SPLINE
SPL {X  -158.491, Y  +370.077, Z    +0.000, E1   +15.910, E3 +25237.550}
SPL {X  -159.771, Y  +383.450, Z    +0.000, E1    +6.314, E3 +25260.705}
SPL {X  -160.000, Y  +392.463, Z    +0.000, E1    +0.112, E3 +25267.212}
SPL {X  -160.000, Y  +399.874, Z    +0.000, E1    -5.508, E3 +25271.714}
SPL {X  -160.000, Y  +411.622, Z    +0.000, E1   -13.815, E3 +25283.834}
SPL {X  -160.000, Y  +419.836, Z    +0.000, E1   -18.198, E3 +25299.008}
SPL {X  -160.000, Y  +430.523, Z    +0.000, E1   -21.710, E3 +25329.208}
SPL {X  -160.000, Y  +433.426, Z    +0.000, E1   -21.735, E3 +25344.623}
SPL {X  -160.000, Y  +436.131, Z    +0.000, E1   -21.710, E3 +25359.098}
SPL {X  -160.000, Y  +439.046, Z    +0.000, E1   -21.732, E3 +25374.591}
SPL {X  -160.000, Y  +442.009, Z    +0.000, E1   -21.719, E3 +25390.413}
SPL {X  -160.000, Y  +444.891, Z    +0.000, E1   -21.724, E3 +25405.769}
SPL {X  -160.000, Y  +449.017, Z    +0.000, E1   -21.792, E3 +25427.560}
SPL {X  -160.000, Y  +452.864, Z    +0.000, E1   -21.730, E3 +25448.178}
SPL {X  -160.000, Y  +455.470, Z    +0.000, E1   -21.722, E3 +25462.067}
SPL {X  -160.000, Y  +458.295, Z    +0.000, E1   -21.738, E3 +25477.088}
SPL {X  -160.000, Y  +461.133, Z    +0.000, E1   -21.720, E3 +25492.271}
SPL {X  -160.000, Y  +464.458, Z    +0.000, E1   -21.770, E3 +25509.789}
SPL {X  -160.000, Y  +468.250, Z    +0.000, E1   -21.764, E3 +25529.943}
SPL {X  -160.000, Y  +472.226, Z    +0.000, E1   -21.782, E3 +25551.101}
SPL {X  -160.000, Y  +476.333, Z    +0.000, E1   -21.767, E3 +25573.015}
SPL {X  -160.000, Y  +480.244, Z    +0.000, E1   -21.765, E3 +25593.880}
SPL {X  -160.000, Y  +484.301, Z    +0.000, E1   -21.775, E3 +25615.408}
SPL {X  -160.000, Y  +488.201, Z    +0.000, E1   -21.768, E3 +25636.168}
SPL {X  -160.000, Y  +492.394, Z    +0.000, E1   -21.802, E3 +25658.343}
SPL {X  -160.000, Y  +496.781, Z    +0.000, E1   -21.798, E3 +25681.654}
SPL {X  -160.000, Y  +501.083, Z    +0.000, E1   -21.796, E3 +25704.584}
SPL {X  -160.000, Y  +504.917, Z    +0.000, E1   -21.764, E3 +25725.088}
SPL {X  -160.000, Y  +508.886, Z    +0.000, E1   -21.791, E3 +25746.174}
SPL {X  -160.000, Y  +513.057, Z    +0.000, E1   -21.767, E3 +25768.482}
SPL {X  -160.000, Y  +517.221, Z    +0.000, E1   -21.778, E3 +25790.635}
SPL {X  -160.000, Y  +521.677, Z    +0.000, E1   -21.781, E3 +25814.396}
SPL {X  -160.000, Y  +525.729, Z    +0.000, E1   -21.753, E3 +25836.035}
SPL {X  -160.000, Y  +529.456, Z    +0.000, E1   -21.766, E3 +25855.815}
SPL {X  -160.000, Y  +533.608, Z    +0.000, E1   -21.776, E3 +25877.945}
SPL {X  -160.000, Y  +538.227, Z    +0.000, E1   -21.794, E3 +25902.477}
SPL {X  -160.000, Y  +542.483, Z    +0.000, E1   -21.764, E3 +25925.203}
SPL {X  -160.000, Y  +546.194, Z    +0.000, E1   -21.754, E3 +25945.019}
SPL {X  -160.000, Y  +550.131, Z    +0.000, E1   -21.771, E3 +25965.955}
SPL {X  -160.000, Y  +554.462, Z    +0.000, E1   -21.777, E3 +25989.009}
SPL {X  -160.000, Y  +558.542, Z    +0.000, E1   -21.758, E3 +26010.782}
SPL {X  -160.000, Y  +562.615, Z    +0.000, E1   -21.776, E3 +26032.437}
SPL {X  -160.000, Y  +566.764, Z    +0.000, E1   -21.764, E3 +26054.562}
SPL {X  -160.000, Y  +570.657, Z    +0.000, E1   -21.758, E3 +26075.310}
SPL {X  -160.000, Y  +574.688, Z    +0.000, E1   -21.771, E3 +26096.752}
SPL {X  -160.000, Y  +578.864, Z    +0.000, E1   -21.770, E3 +26119.003}
SPL {X  -160.000, Y  +582.807, Z    +0.000, E1   -21.754, E3 +26140.057}
SPL {X  -160.000, Y  +586.993, Z    +0.000, E1   -21.779, E3 +26162.293}
SPL {X  -160.000, Y  +591.368, Z    +0.000, E1   -21.775, E3 +26185.580}
SPL {X  -160.000, Y  +595.703, Z    +0.000, E1   -21.775, E3 +26208.690}
SPL {X  -160.000, Y  +599.558, Z    +0.000, E1   -21.748, E3 +26229.267}
SPL {X  -160.000, Y  +603.126, Z    +0.000, E1   -21.757, E3 +26248.247}
SPL {X  -160.000, Y  +607.107, Z    +0.000, E1   -21.766, E3 +26269.472}
SPL {X  -160.000, Y  +611.246, Z    +0.000, E1   -21.760, E3 +26291.545}
SPL {X  -160.000, Y  +615.151, Z    +0.000, E1   -21.752, E3 +26312.358}
SPL {X  -160.000, Y  +618.728, Z    +0.000, E1   -21.747, E3 +26331.421}
SPL {X  -160.000, Y  +622.318, Z    +0.000, E1   -21.753, E3 +26350.535}
SPL {X  -160.000, Y  +625.877, Z    +0.000, E1   -21.745, E3 +26369.514}
SPL {X  -160.000, Y  +629.892, Z    +0.000, E1   -21.777, E3 +26390.837}
SPL {X  -160.000, Y  +634.024, Z    +0.000, E1   -21.756, E3 +26412.888}
SPL {X  -160.000, Y  +637.661, Z    +0.000, E1   -21.748, E3 +26432.278}
SPL {X  -160.000, Y  +641.244, Z    +0.000, E1   -21.752, E3 +26451.349}
SPL {X  -160.000, Y  +645.120, Z    +0.000, E1   -21.762, E3 +26471.981}
SPL {X  -160.000, Y  +649.214, Z    +0.000, E1   -21.766, E3 +26493.770}
SPL {X  -160.000, Y  +653.188, Z    +0.000, E1   -21.771, E3 +26514.832}
SPL {X  -160.000, Y  +656.905, Z    +0.000, E1   -21.769, E3 +26534.607}
SPL {X  -160.000, Y  +660.685, Z    +0.000, E1   -21.769, E3 +26554.775}
SPL {X  -160.000, Y  +664.985, Z    +0.000, E1   -21.790, E3 +26577.628}
SPL {X  -159.993, Y  +669.170, Z    +0.000, E1   -21.763, E3 +26599.987}
SPL {X  -159.916, Y  +672.869, Z    +0.000, E1   -21.755, E3 +26619.732}
SPL {X  -159.752, Y  +676.610, Z    +0.000, E1   -21.740, E3 +26639.806}
SPL {X  -159.478, Y  +680.618, Z    +0.000, E1   -21.719, E3 +26661.406}
SPL {X  -159.108, Y  +684.576, Z    +0.000, E1   -21.664, E3 +26682.875}
SPL {X  -158.638, Y  +688.530, Z    +0.000, E1   -21.617, E3 +26704.396}
SPL {X  -158.097, Y  +692.303, Z    +0.000, E1   -21.529, E3 +26725.114}
ENDSPLINE

SPLINE
SPL {X  -158.264, Y  +691.203, Z    +0.000, E1   -17.264, E3 +26761.859}
SPL {X  -159.000, Y  +685.560, Z    +0.000, E1   -12.398, E3 +26783.035}
SPL {X  -159.924, Y  +672.625, Z    +0.000, E1    -3.689, E3 +26798.052}
SPL {X  -160.000, Y  +663.203, Z    +0.000, E1    +3.155, E3 +26804.706}
SPL {X  -160.000, Y  +652.103, Z    +0.000, E1   +11.247, E3 +26816.377}
SPL {X  -160.000, Y  +641.822, Z    +0.000, E1   +17.059, E3 +26835.750}
SPL {X  -160.000, Y  +631.293, Z    +0.000, E1   +20.354, E3 +26869.630}
SPL {X  -160.000, Y  +627.542, Z    +0.000, E1   +20.380, E3 +26891.037}
SPL {X  -160.000, Y  +623.532, Z    +0.000, E1   +20.378, E3 +26914.003}
SPL {X  -160.000, Y  +619.329, Z    +0.000, E1   +20.391, E3 +26938.040}
SPL {X  -160.000, Y  +614.967, Z    +0.000, E1   +20.392, E3 +26963.020}
SPL {X  -160.000, Y  +611.206, Z    +0.000, E1   +20.351, E3 +26984.692}
SPL {X  -160.000, Y  +607.824, Z    +0.000, E1   +20.354, E3 +27004.112}
SPL {X  -160.000, Y  +603.899, Z    +0.000, E1   +20.373, E3 +27026.563}
SPL {X  -160.000, Y  +599.617, Z    +0.000, E1   +20.384, E3 +27051.056}
SPL {X  -160.000, Y  +595.532, Z    +0.000, E1   +20.373, E3 +27074.417}
SPL {X  -160.000, Y  +591.705, Z    +0.000, E1   +20.373, E3 +27096.342}
SPL {X  -160.000, Y  +588.037, Z    +0.000, E1   +20.359, E3 +27117.428}
SPL {X  -160.000, Y  +584.320, Z    +0.000, E1   +20.364, E3 +27138.730}
SPL {X  -160.000, Y  +580.616, Z    +0.000, E1   +20.357, E3 +27159.957}
SPL {X  -160.000, Y  +577.083, Z    +0.000, E1   +20.358, E3 +27180.205}
SPL {X  -160.000, Y  +573.158, Z    +0.000, E1   +20.377, E3 +27202.658}
SPL {X  -160.000, Y  +568.802, Z    +0.000, E1   +20.385, E3 +27227.609}
SPL {X  -160.000, Y  +564.937, Z    +0.000, E1   +20.350, E3 +27249.830}
SPL {X  -160.000, Y  +561.213, Z    +0.000, E1   +20.372, E3 +27271.116}
SPL {X  -160.000, Y  +557.320, Z    +0.000, E1   +20.363, E3 +27293.443}
SPL {X  -160.000, Y  +553.712, Z    +0.000, E1   +20.355, E3 +27314.143}
SPL {X  -160.000, Y  +550.040, Z    +0.000, E1   +20.360, E3 +27335.181}
SPL {X  -160.000, Y  +546.180, Z    +0.000, E1   +20.370, E3 +27357.236}
SPL {X  -160.000, Y  +542.032, Z    +0.000, E1   +20.384, E3 +27380.975}
SPL {X  -160.000, Y  +537.870, Z    +0.000, E1   +20.372, E3 +27404.851}
SPL {X  -160.000, Y  +534.086, Z    +0.000, E1   +20.356, E3 +27426.605}
SPL {X  -160.000, Y  +530.164, Z    +0.000, E1   +20.382, E3 +27448.954}
SPL {X  -160.000, Y  +527.505, Z    +0.000, E1   +20.318, E3 +27464.328}
SPL {X  -160.000, Y  +511.620, Z    +0.000, E1   +28.365, E3 +27474.791}
SPL {X  -160.000, Y  +507.906, Z    +0.000, E1   +28.152, E3 +27491.186}
SPL {X  -160.000, Y  +506.085, Z    +0.000, E1   +26.146, E3 +27513.646}
SPL {X  -160.000, Y  +504.342, Z    +0.000, E1   +24.109, E3 +27537.161}
SPL {X  -160.000, Y  +503.002, Z    +0.000, E1   +22.325, E3 +27558.166}
SPL {X  -160.000, Y  +500.783, Z    +0.000, E1   +21.421, E3 +27577.756}
SPL {X  -160.000, Y  +497.229, Z    +0.000, E1   +21.403, E3 +27597.064}
SPL {X  -160.000, Y  +493.901, Z    +0.000, E1   +21.409, E3 +27615.083}
SPL {X  -160.000, Y  +490.791, Z    +0.000, E1   +21.400, E3 +27631.956}
SPL {X  -160.000, Y  +487.647, Z    +0.000, E1   +21.401, E3 +27649.002}
SPL {X  -160.000, Y  +484.273, Z    +0.000, E1   +21.408, E3 +27667.282}
SPL {X  -160.000, Y  +481.093, Z    +0.000, E1   +21.389, E3 +27684.591}
SPL {X  -160.000, Y  +478.021, Z    +0.000, E1   +21.401, E3 +27701.198}
SPL {X  -160.000, Y  +474.639, Z    +0.000, E1   +21.410, E3 +27719.489}
SPL {X  -160.000, Y  +471.343, Z    +0.000, E1   +21.399, E3 +27737.391}
SPL {X  -160.000, Y  +468.133, Z    +0.000, E1   +21.402, E3 +27754.782}
SPL {X  -160.000, Y  +464.638, Z    +0.000, E1   +21.421, E3 +27773.632}
SPL {X  -160.000, Y  +461.045, Z    +0.000, E1   +21.424, E3 +27793.045}
SPL {X  -160.000, Y  +457.606, Z    +0.000, E1   +21.413, E3 +27811.755}
SPL {X  -160.000, Y  +454.417, Z    +0.000, E1   +21.401, E3 +27829.064}
SPL {X  -160.000, Y  +451.425, Z    +0.000, E1   +21.404, E3 +27845.286}
SPL {X  -160.000, Y  +448.039, Z    +0.000, E1   +21.417, E3 +27863.578}
SPL {X  -160.000, Y  +444.787, Z    +0.000, E1   +21.414, E3 +27881.134}
SPL {X  -160.000, Y  +441.637, Z    +0.000, E1   +21.431, E3 +27898.112}
SPL {X  -160.000, Y  +438.199, Z    +0.000, E1   +21.432, E3 +27916.716}
SPL {X  -160.000, Y  +434.875, Z    +0.000, E1   +21.424, E3 +27934.756}
SPL {X  -160.000, Y  +431.689, Z    +0.000, E1   +21.423, E3 +27952.004}
SPL {X  -160.000, Y  +428.451, Z    +0.000, E1   +21.430, E3 +27969.483}
SPL {X  -160.000, Y  +425.120, Z    +0.000, E1   +21.430, E3 +27987.548}
SPL {X  -160.000, Y  +421.671, Z    +0.000, E1   +21.430, E3 +28006.232}
SPL {X  -160.000, Y  +418.225, Z    +0.000, E1   +21.425, E3 +28024.913}
SPL {X  -160.000, Y  +414.956, Z    +0.000, E1   +21.424, E3 +28042.594}
SPL {X  -160.000, Y  +411.834, Z    +0.000, E1   +21.420, E3 +28059.512}
SPL {X  -160.000, Y  +408.570, Z    +0.000, E1   +21.432, E3 +28077.121}
SPL {X  -160.000, Y  +405.237, Z    +0.000, E1   +21.432, E3 +28095.150}
SPL {X  -160.000, Y  +402.004, Z    +0.000, E1   +21.424, E3 +28112.725}
SPL {X  -160.000, Y  +398.626, Z    +0.000, E1   +21.425, E3 +28131.031}
SPL {X  -160.000, Y  +395.405, Z    +0.000, E1   +21.422, E3 +28148.449}
SPL {X  -160.000, Y  +392.641, Z    +0.000, E1   +21.407, E3 +28163.447}
SPL {X  -159.989, Y  +390.129, Z    +0.000, E1   +21.406, E3 +28177.088}
SPL {X  -159.932, Y  +387.337, Z    +0.000, E1   +21.403, E3 +28192.284}
SPL {X  -159.823, Y  +384.478, Z    +0.000, E1   +21.379, E3 +28207.947}
SPL {X  -159.660, Y  +381.581, Z    +0.000, E1   +21.363, E3 +28223.835}
SPL {X  -159.452, Y  +378.773, Z    +0.000, E1   +21.330, E3 +28239.282}
SPL {X  -159.222, Y  +376.244, Z    +0.000, E1   +21.297, E3 +28253.244}
SPL {X  -158.814, Y  +372.556, Z    +0.000, E1   +21.316, E3 +28273.511}
SPL {X  -158.301, Y  +368.743, Z    +0.000, E1   +21.199, E3 +28294.833}
SPL {X  -157.981, Y  +366.660, Z    +0.000, E1   +19.986, E3 +28317.800}
ENDSPLINE

SPLINE
SPL {X  -158.491, Y  +370.077, Z    +0.000, E1   +15.910, E3 +28342.814}
SPL {X  -159.771, Y  +383.450, Z    +0.000, E1    +6.314, E3 +28365.969}
SPL {X  -160.000, Y  +392.463, Z    +0.000, E1    +0.112, E3 +28372.476}
SPL {X  -160.000, Y  +399.874, Z    +0.000, E1    -5.508, E3 +28376.978}
SPL {X  -160.000, Y  +411.622, Z    +0.000, E1   -13.815, E3 +28389.098}
SPL {X  -160.000, Y  +419.836, Z    +0.000, E1   -18.198, E3 +28404.272}
SPL {X  -160.000, Y  +430.523, Z    +0.000, E1   -21.710, E3 +28434.472}
SPL {X  -160.000, Y  +433.426, Z    +0.000, E1   -21.735, E3 +28449.886}
SPL {X  -160.000, Y  +436.131, Z    +0.000, E1   -21.710, E3 +28464.361}
SPL {X  -160.000, Y  +439.046, Z    +0.000, E1   -21.732, E3 +28479.854}
SPL {X  -160.000, Y  +442.009, Z    +0.000, E1   -21.719, E3 +28495.676}
SPL {X  -160.000, Y  +444.891, Z    +0.000, E1   -21.724, E3 +28511.032}
SPL {X  -160.000, Y  +449.017, Z    +0.000, E1   -21.792, E3 +28532.824}
SPL {X  -160.000, Y  +452.864, Z    +0.000, E1   -21.730, E3 +28553.442}
SPL {X  -160.000, Y  +455.470, Z    +0.000, E1   -21.722, E3 +28567.331}
SPL {X  -160.000, Y  +458.295, Z    +0.000, E1   -21.738, E3 +28582.351}
SPL {X  -160.000, Y  +461.133, Z    +0.000, E1   -21.720, E3 +28597.534}
SPL {X  -160.000, Y  +464.458, Z    +0.000, E1   -21.770, E3 +28615.053}
SPL {X  -160.000, Y  +468.250, Z    +0.000, E1   -21.764, E3 +28635.206}
SPL {X  -160.000, Y  +472.226, Z    +0.000, E1   -21.782, E3 +28656.364}
SPL {X  -160.000, Y  +476.333, Z    +0.000, E1   -21.767, E3 +28678.279}
SPL {X  -160.000, Y  +480.244, Z    +0.000, E1   -21.765, E3 +28699.143}
SPL {X  -160.000, Y  +484.301, Z    +0.000, E1   -21.775, E3 +28720.672}
SPL {X  -160.000, Y  +488.201, Z    +0.000, E1   -21.768, E3 +28741.432}
SPL {X  -160.000, Y  +492.394, Z    +0.000, E1   -21.802, E3 +28763.606}
SPL {X  -160.000, Y  +496.781, Z    +0.000, E1   -21.798, E3 +28786.917}
SPL {X  -160.000, Y  +501.083, Z    +0.000, E1   -21.796, E3 +28809.847}
SPL {X  -160.000, Y  +504.917, Z    +0.000, E1   -21.764, E3 +28830.352}
SPL {X  -160.000, Y  +508.886, Z    +0.000, E1   -21.791, E3 +28851.438}
SPL {X  -160.000, Y  +513.057, Z    +0.000, E1   -21.767, E3 +28873.746}
SPL {X  -160.000, Y  +517.221, Z    +0.000, E1   -21.778, E3 +28895.898}
SPL {X  -160.000, Y  +521.677, Z    +0.000, E1   -21.781, E3 +28919.659}
SPL {X  -160.000, Y  +525.729, Z    +0.000, E1   -21.753, E3 +28941.299}
SPL {X  -160.000, Y  +529.456, Z    +0.000, E1   -21.766, E3 +28961.078}
SPL {X  -160.000, Y  +533.608, Z    +0.000, E1   -21.776, E3 +28983.209}
SPL {X  -160.000, Y  +538.227, Z    +0.000, E1   -21.794, E3 +29007.741}
SPL {X  -160.000, Y  +542.483, Z    +0.000, E1   -21.764, E3 +29030.466}
SPL {X  -160.000, Y  +546.194, Z    +0.000, E1   -21.754, E3 +29050.283}
SPL {X  -160.000, Y  +550.131, Z    +0.000, E1   -21.771, E3 +29071.218}
SPL {X  -160.000, Y  +554.462, Z    +0.000, E1   -21.777, E3 +29094.272}
SPL {X  -160.000, Y  +558.542, Z    +0.000, E1   -21.758, E3 +29116.045}
SPL {X  -160.000, Y  +562.615, Z    +0.000, E1   -21.776, E3 +29137.701}
SPL {X  -160.000, Y  +566.764, Z    +0.000, E1   -21.764, E3 +29159.826}
SPL {X  -160.000, Y  +570.657, Z    +0.000, E1   -21.758, E3 +29180.573}
SPL {X  -160.000, Y  +574.688, Z    +0.000, E1   -21.771, E3 +29202.016}
SPL {X  -160.000, Y  +578.864, Z    +0.000, E1   -21.770, E3 +29224.267}
SPL {X  -160.000, Y  +582.807, Z    +0.000, E1   -21.754, E3 +29245.321}
SPL {X  -160.000, Y  +586.993, Z    +0.000, E1   -21.779, E3 +29267.557}
SPL {X  -160.000, Y  +591.368, Z    +0.000, E1   -21.775, E3 +29290.844}
SPL {X  -160.000, Y  +595.703, Z    +0.000, E1   -21.775, E3 +29313.953}
SPL {X  -160.000, Y  +599.558, Z    +0.000, E1   -21.748, E3 +29334.530}
SPL {X  -160.000, Y  +603.126, Z    +0.000, E1   -21.757, E3 +29353.510}
SPL {X  -160.000, Y  +607.107, Z    +0.000, E1   -21.766, E3 +29374.735}
SPL {X  -160.000, Y  +611.246, Z    +0.000, E1   -21.760, E3 +29396.808}
SPL {X  -160.000, Y  +615.151, Z    +0.000, E1   -21.752, E3 +29417.622}
SPL {X  -160.000, Y  +618.728, Z    +0.000, E1   -21.747, E3 +29436.684}
SPL {X  -160.000, Y  +622.318, Z    +0.000, E1   -21.753, E3 +29455.799}
SPL {X  -160.000, Y  +625.877, Z    +0.000, E1   -21.745, E3 +29474.777}
SPL {X  -160.000, Y  +629.892, Z    +0.000, E1   -21.777, E3 +29496.101}
SPL {X  -160.000, Y  +634.024, Z    +0.000, E1   -21.756, E3 +29518.151}
SPL {X  -160.000, Y  +637.661, Z    +0.000, E1   -21.748, E3 +29537.542}
SPL {X  -160.000, Y  +641.244, Z    +0.000, E1   -21.752, E3 +29556.612}
SPL {X  -160.000, Y  +645.120, Z    +0.000, E1   -21.762, E3 +29577.245}
SPL {X  -160.000, Y  +649.214, Z    +0.000, E1   -21.766, E3 +29599.033}
SPL {X  -160.000, Y  +653.188, Z    +0.000, E1   -21.771, E3 +29620.096}
SPL {X  -160.000, Y  +656.905, Z    +0.000, E1   -21.769, E3 +29639.871}
SPL {X  -160.000, Y  +660.685, Z    +0.000, E1   -21.769, E3 +29660.039}
SPL {X  -160.000, Y  +664.985, Z    +0.000, E1   -21.790, E3 +29682.892}
SPL {X  -159.993, Y  +669.170, Z    +0.000, E1   -21.763, E3 +29705.250}
SPL {X  -159.916, Y  +672.869, Z    +0.000, E1   -21.755, E3 +29724.995}
SPL {X  -159.752, Y  +676.610, Z    +0.000, E1   -21.740, E3 +29745.070}
SPL {X  -159.478, Y  +680.618, Z    +0.000, E1   -21.719, E3 +29766.669}
SPL {X  -159.108, Y  +684.576, Z    +0.000, E1   -21.664, E3 +29788.138}
SPL {X  -158.638, Y  +688.530, Z    +0.000, E1   -21.617, E3 +29809.660}
SPL {X  -158.097, Y  +692.303, Z    +0.000, E1   -21.529, E3 +29830.378}
ENDSPLINE

SPLINE
SPL {X  -158.264, Y  +691.203, Z    +0.000, E1   -17.264, E3 +29867.123}
SPL {X  -159.000, Y  +685.560, Z    +0.000, E1   -12.398, E3 +29888.298}
SPL {X  -159.924, Y  +672.625, Z    +0.000, E1    -3.689, E3 +29903.316}
SPL {X  -160.000, Y  +663.203, Z    +0.000, E1    +3.155, E3 +29909.970}
SPL {X  -160.000, Y  +652.103, Z    +0.000, E1   +11.247, E3 +29921.640}
SPL {X  -160.000, Y  +641.822, Z    +0.000, E1   +17.059, E3 +29941.014}
SPL {X  -160.000, Y  +631.293, Z    +0.000, E1   +20.354, E3 +29974.893}
SPL {X  -160.000, Y  +627.542, Z    +0.000, E1   +20.380, E3 +29996.300}
SPL {X  -160.000, Y  +623.532, Z    +0.000, E1   +20.378, E3 +30019.266}
SPL {X  -160.000, Y  +619.329, Z    +0.000, E1   +20.391, E3 +30043.304}
SPL {X  -160.000, Y  +614.967, Z    +0.000, E1   +20.392, E3 +30068.283}
SPL {X  -160.000, Y  +611.206, Z    +0.000, E1   +20.351, E3 +30089.955}
SPL {X  -160.000, Y  +607.824, Z    +0.000, E1   +20.354, E3 +30109.376}
SPL {X  -160.000, Y  +603.899, Z    +0.000, E1   +20.373, E3 +30131.826}
SPL {X  -160.000, Y  +599.617, Z    +0.000, E1   +20.384, E3 +30156.320}
SPL {X  -160.000, Y  +595.532, Z    +0.000, E1   +20.373, E3 +30179.680}
SPL {X  -160.000, Y  +591.705, Z    +0.000, E1   +20.373, E3 +30201.605}
SPL {X  -160.000, Y  +588.037, Z    +0.000, E1   +20.359, E3 +30222.692}
SPL {X  -160.000, Y  +584.320, Z    +0.000, E1   +20.364, E3 +30243.994}
SPL {X  -160.000, Y  +580.616, Z    +0.000, E1   +20.357, E3 +30265.220}
SPL {X  -160.000, Y  +577.083, Z    +0.000, E1   +20.358, E3 +30285.469}
SPL {X  -160.000, Y  +573.158, Z    +0.000, E1   +20.377, E3 +30307.921}
SPL {X  -160.000, Y  +568.802, Z    +0.000, E1   +20.385, E3 +30332.873}
SPL {X  -160.000, Y  +564.937, Z    +0.000, E1   +20.350, E3 +30355.094}
SPL {X  -160.000, Y  +561.213, Z    +0.000, E1   +20.372, E3 +30376.380}
SPL {X  -160.000, Y  +557.320, Z    +0.000, E1   +20.363, E3 +30398.707}
SPL {X  -160.000, Y  +553.712, Z    +0.000, E1   +20.355, E3 +30419.406}
SPL {X  -160.000, Y  +550.040, Z    +0.000, E1   +20.360, E3 +30440.444}
SPL {X  -160.000, Y  +546.180, Z    +0.000, E1   +20.370, E3 +30462.500}
SPL {X  -160.000, Y  +542.032, Z    +0.000, E1   +20.384, E3 +30486.239}
SPL {X  -160.000, Y  +537.870, Z    +0.000, E1   +20.372, E3 +30510.115}
SPL {X  -160.000, Y  +534.086, Z    +0.000, E1   +20.356, E3 +30531.868}
SPL {X  -160.000, Y  +530.164, Z    +0.000, E1   +20.382, E3 +30554.218}
SPL {X  -160.000, Y  +527.505, Z    +0.000, E1   +20.318, E3 +30569.592}
SPL {X  -160.000, Y  +511.620, Z    +0.000, E1   +28.365, E3 +30580.055}
SPL {X  -160.000, Y  +507.906, Z    +0.000, E1   +28.152, E3 +30596.450}
SPL {X  -160.000, Y  +506.085, Z    +0.000, E1   +26.146, E3 +30618.909}
SPL {X  -160.000, Y  +504.342, Z    +0.000, E1   +24.109, E3 +30642.424}
SPL {X  -160.000, Y  +503.002, Z    +0.000, E1   +22.325, E3 +30663.430}
SPL {X  -160.000, Y  +500.783, Z    +0.000, E1   +21.421, E3 +30683.019}
SPL {X  -160.000, Y  +497.229, Z    +0.000, E1   +21.403, E3 +30702.327}
SPL {X  -160.000, Y  +493.901, Z    +0.000, E1   +21.409, E3 +30720.346}
SPL {X  -160.000, Y  +490.791, Z    +0.000, E1   +21.400, E3 +30737.219}
SPL {X  -160.000, Y  +487.647, Z    +0.000, E1   +21.401, E3 +30754.265}
SPL {X  -160.000, Y  +484.273, Z    +0.000, E1   +21.408, E3 +30772.545}
SPL {X  -160.000, Y  +481.093, Z    +0.000, E1   +21.389, E3 +30789.854}
SPL {X  -160.000, Y  +478.021, Z    +0.000, E1   +21.401, E3 +30806.461}
SPL {X  -160.000, Y  +474.639, Z    +0.000, E1   +21.410, E3 +30824.752}
SPL {X  -160.000, Y  +471.343, Z    +0.000, E1   +21.399, E3 +30842.654}
SPL {X  -160.000, Y  +468.133, Z    +0.000, E1   +21.402, E3 +30860.046}
SPL {X  -160.000, Y  +464.638, Z    +0.000, E1   +21.421, E3 +30878.895}
SPL {X  -160.000, Y  +461.045, Z    +0.000, E1   +21.424, E3 +30898.309}
SPL {X  -160.000, Y  +457.606, Z    +0.000, E1   +21.413, E3 +30917.019}
SPL {X  -160.000, Y  +454.417, Z    +0.000, E1   +21.401, E3 +30934.328}
SPL {X  -160.000, Y  +451.425, Z    +0.000, E1   +21.404, E3 +30950.549}
SPL {X  -160.000, Y  +448.039, Z    +0.000, E1   +21.417, E3 +30968.842}
SPL {X  -160.000, Y  +444.787, Z    +0.000, E1   +21.414, E3 +30986.397}
SPL {X  -160.000, Y  +441.637, Z    +0.000, E1   +21.431, E3 +31003.375}
SPL {X  -160.000, Y  +438.199, Z    +0.000, E1   +21.432, E3 +31021.979}
SPL {X  -160.000, Y  +434.875, Z    +0.000, E1   +21.424, E3 +31040.019}
SPL {X  -160.000, Y  +431.689, Z    +0.000, E1   +21.423, E3 +31057.267}
SPL {X  -160.000, Y  +428.451, Z    +0.000, E1   +21.430, E3 +31074.747}
SPL {X  -160.000, Y  +425.120, Z    +0.000, E1   +21.430, E3 +31092.811}
SPL {X  -160.000, Y  +421.671, Z    +0.000, E1   +21.430, E3 +31111.495}
SPL {X  -160.000, Y  +418.225, Z    +0.000, E1   +21.425, E3 +31130.177}
SPL {X  -160.000, Y  +414.956, Z    +0.000, E1   +21.424, E3 +31147.858}
SPL {X  -160.000, Y  +411.834, Z    +0.000, E1   +21.420, E3 +31164.776}
SPL {X  -160.000, Y  +408.570, Z    +0.000, E1   +21.432, E3 +31182.385}
SPL {X  -160.000, Y  +405.237, Z    +0.000, E1   +21.432, E3 +31200.413}
SPL {X  -160.000, Y  +402.004, Z    +0.000, E1   +21.424, E3 +31217.989}
SPL {X  -160.000, Y  +398.626, Z    +0.000, E1   +21.425, E3 +31236.295}
SPL {X  -160.000, Y  +395.405, Z    +0.000, E1   +21.422, E3 +31253.712}
SPL {X  -160.000, Y  +392.641, Z    +0.000, E1   +21.407, E3 +31268.710}
SPL {X  -159.989, Y  +390.129, Z    +0.000, E1   +21.406, E3 +31282.351}
SPL {X  -159.932, Y  +387.337, Z    +0.000, E1   +21.403, E3 +31297.547}
SPL {X  -159.823, Y  +384.478, Z    +0.000, E1   +21.379, E3 +31313.210}
SPL {X  -159.660, Y  +381.581, Z    +0.000, E1   +21.363, E3 +31329.098}
SPL {X  -159.452, Y  +378.773, Z    +0.000, E1   +21.330, E3 +31344.545}
SPL {X  -159.222, Y  +376.244, Z    +0.000, E1   +21.297, E3 +31358.507}
SPL {X  -158.814, Y  +372.556, Z    +0.000, E1   +21.316, E3 +31378.775}
SPL {X  -158.301, Y  +368.743, Z    +0.000, E1   +21.199, E3 +31400.096}
SPL {X  -157.981, Y  +366.660, Z    +0.000, E1   +19.986, E3 +31423.064}
ENDSPLINE

SPLINE
SPL {X  -158.491, Y  +370.077, Z    +0.000, E1   +15.910, E3 +31448.077}
SPL {X  -159.771, Y  +383.450, Z    +0.000, E1    +6.314, E3 +31471.232}
SPL {X  -160.000, Y  +392.463, Z    +0.000, E1    +0.112, E3 +31477.739}
SPL {X  -160.000, Y  +399.874, Z    +0.000, E1    -5.508, E3 +31482.242}
SPL {X  -160.000, Y  +411.622, Z    +0.000, E1   -13.815, E3 +31494.361}
SPL {X  -160.000, Y  +419.836, Z    +0.000, E1   -18.198, E3 +31509.535}
SPL {X  -160.000, Y  +430.523, Z    +0.000, E1   -21.710, E3 +31539.735}
SPL {X  -160.000, Y  +433.426, Z    +0.000, E1   -21.735, E3 +31555.150}
SPL {X  -160.000, Y  +436.131, Z    +0.000, E1   -21.710, E3 +31569.625}
SPL {X  -160.000, Y  +439.046, Z    +0.000, E1   -21.732, E3 +31585.118}
SPL {X  -160.000, Y  +442.009, Z    +0.000, E1   -21.719, E3 +31600.940}
SPL {X  -160.000, Y  +444.891, Z    +0.000, E1   -21.724, E3 +31616.296}
SPL {X  -160.000, Y  +449.017, Z    +0.000, E1   -21.792, E3 +31638.087}
SPL {X  -160.000, Y  +452.864, Z    +0.000, E1   -21.730, E3 +31658.705}
SPL {X  -160.000, Y  +455.470, Z    +0.000, E1   -21.722, E3 +31672.594}
SPL {X  -160.000, Y  +458.295, Z    +0.000, E1   -21.738, E3 +31687.615}
SPL {X  -160.000, Y  +461.133, Z    +0.000, E1   -21.720, E3 +31702.798}
SPL {X  -160.000, Y  +464.458, Z    +0.000, E1   -21.770, E3 +31720.316}
SPL {X  -160.000, Y  +468.250, Z    +0.000, E1   -21.764, E3 +31740.470}
SPL {X  -160.000, Y  +472.226, Z    +0.000, E1   -21.782, E3 +31761.628}
SPL {X  -160.000, Y  +476.333, Z    +0.000, E1   -21.767, E3 +31783.543}
SPL {X  -160.000, Y  +480.244, Z    +0.000, E1   -21.765, E3 +31804.407}
SPL {X  -160.000, Y  +484.301, Z    +0.000, E1   -21.775, E3 +31825.935}
SPL {X  -160.000, Y  +488.201, Z    +0.000, E1   -21.768, E3 +31846.695}
SPL {X  -160.000, Y  +492.394, Z    +0.000, E1   -21.802, E3 +31868.870}
SPL {X  -160.000, Y  +496.781, Z    +0.000, E1   -21.798, E3 +31892.181}
SPL {X  -160.000, Y  +501.083, Z    +0.000, E1   -21.796, E3 +31915.111}
SPL {X  -160.000, Y  +504.917, Z    +0.000, E1   -21.764, E3 +31935.615}
SPL {X  -160.000, Y  +508.886, Z    +0.000, E1   -21.791, E3 +31956.702}
SPL {X  -160.000, Y  +513.057, Z    +0.000, E1   -21.767, E3 +31979.009}
SPL {X  -160.000, Y  +517.221, Z    +0.000, E1   -21.778, E3 +32001.162}
SPL {X  -160.000, Y  +521.677, Z    +0.000, E1   -21.781, E3 +32024.923}
SPL {X  -160.000, Y  +525.729, Z    +0.000, E1   -21.753, E3 +32046.562}
SPL {X  -160.000, Y  +529.456, Z    +0.000, E1   -21.766, E3 +32066.342}
SPL {X  -160.000, Y  +533.608, Z    +0.000, E1   -21.776, E3 +32088.472}
SPL {X  -160.000, Y  +538.227, Z    +0.000, E1   -21.794, E3 +32113.004}
SPL {X  -160.000, Y  +542.483, Z    +0.000, E1   -21.764, E3 +32135.730}
SPL {X  -160.000, Y  +546.194, Z    +0.000, E1   -21.754, E3 +32155.546}
SPL {X  -160.000, Y  +550.131, Z    +0.000, E1   -21.771, E3 +32176.482}
SPL {X  -160.000, Y  +554.462, Z    +0.000, E1   -21.777, E3 +32199.536}
SPL {X  -160.000, Y  +558.542, Z    +0.000, E1   -21.758, E3 +32221.309}
SPL {X  -160.000, Y  +562.615, Z    +0.000, E1   -21.776, E3 +32242.964}
SPL {X  -160.000, Y  +566.764, Z    +0.000, E1   -21.764, E3 +32265.089}
SPL {X  -160.000, Y  +570.657, Z    +0.000, E1   -21.758, E3 +32285.837}
SPL {X  -160.000, Y  +574.688, Z    +0.000, E1   -21.771, E3 +32307.279}
SPL {X  -160.000, Y  +578.864, Z    +0.000, E1   -21.770, E3 +32329.530}
SPL {X  -160.000, Y  +582.807, Z    +0.000, E1   -21.754, E3 +32350.584}
SPL {X  -160.000, Y  +586.993, Z    +0.000, E1   -21.779, E3 +32372.820}
SPL {X  -160.000, Y  +591.368, Z    +0.000, E1   -21.775, E3 +32396.107}
SPL {X  -160.000, Y  +595.703, Z    +0.000, E1   -21.775, E3 +32419.217}
SPL {X  -160.000, Y  +599.558, Z    +0.000, E1   -21.748, E3 +32439.794}
SPL {X  -160.000, Y  +603.126, Z    +0.000, E1   -21.757, E3 +32458.774}
SPL {X  -160.000, Y  +607.107, Z    +0.000, E1   -21.766, E3 +32479.999}
SPL {X  -160.000, Y  +611.246, Z    +0.000, E1   -21.760, E3 +32502.072}
SPL {X  -160.000, Y  +615.151, Z    +0.000, E1   -21.752, E3 +32522.885}
SPL {X  -160.000, Y  +618.728, Z    +0.000, E1   -21.747, E3 +32541.948}
SPL {X  -160.000, Y  +622.318, Z    +0.000, E1   -21.753, E3 +32561.062}
SPL {X  -160.000, Y  +625.877, Z    +0.000, E1   -21.745, E3 +32580.041}
SPL {X  -160.000, Y  +629.892, Z    +0.000, E1   -21.777, E3 +32601.364}
SPL {X  -160.000, Y  +634.024, Z    +0.000, E1   -21.756, E3 +32623.415}
SPL {X  -160.000, Y  +637.661, Z    +0.000, E1   -21.748, E3 +32642.805}
SPL {X  -160.000, Y  +641.244, Z    +0.000, E1   -21.752, E3 +32661.876}
SPL {X  -160.000, Y  +645.120, Z    +0.000, E1   -21.762, E3 +32682.508}
SPL {X  -160.000, Y  +649.214, Z    +0.000, E1   -21.766, E3 +32704.297}
SPL {X  -160.000, Y  +653.188, Z    +0.000, E1   -21.771, E3 +32725.359}
SPL {X  -160.000, Y  +656.905, Z    +0.000, E1   -21.769, E3 +32745.134}
SPL {X  -160.000, Y  +660.685, Z    +0.000, E1   -21.769, E3 +32765.302}
SPL {X  -160.000, Y  +664.985, Z    +0.000, E1   -21.790, E3 +32788.155}
SPL {X  -159.993, Y  +669.170, Z    +0.000, E1   -21.763, E3 +32810.514}
SPL {X  -159.916, Y  +672.869, Z    +0.000, E1   -21.755, E3 +32830.259}
SPL {X  -159.752, Y  +676.610, Z    +0.000, E1   -21.740, E3 +32850.333}
SPL {X  -159.478, Y  +680.618, Z    +0.000, E1   -21.719, E3 +32871.933}
SPL {X  -159.108, Y  +684.576, Z    +0.000, E1   -21.664, E3 +32893.402}
SPL {X  -158.638, Y  +688.530, Z    +0.000, E1   -21.617, E3 +32914.923}
SPL {X  -158.097, Y  +692.303, Z    +0.000, E1   -21.529, E3 +32935.641}
ENDSPLINE

SPLINE
SPL {X  -158.264, Y  +691.203, Z    +0.000, E1   -17.264, E3 +32972.387}
SPL {X  -159.000, Y  +685.560, Z    +0.000, E1   -12.398, E3 +32993.562}
SPL {X  -159.924, Y  +672.625, Z    +0.000, E1    -3.689, E3 +33008.579}
SPL {X  -160.000, Y  +663.203, Z    +0.000, E1    +3.155, E3 +33015.234}
SPL {X  -160.000, Y  +652.103, Z    +0.000, E1   +11.247, E3 +33026.904}
SPL {X  -160.000, Y  +641.822, Z    +0.000, E1   +17.059, E3 +33046.277}
SPL {X  -160.000, Y  +631.293, Z    +0.000, E1   +20.354, E3 +33080.157}
SPL {X  -160.000, Y  +627.542, Z    +0.000, E1   +20.380, E3 +33101.564}
SPL {X  -160.000, Y  +623.532, Z    +0.000, E1   +20.378, E3 +33124.530}
SPL {X  -160.000, Y  +619.329, Z    +0.000, E1   +20.391, E3 +33148.567}
SPL {X  -160.000, Y  +614.967, Z    +0.000, E1   +20.392, E3 +33173.547}
SPL {X  -160.000, Y  +611.206, Z    +0.000, E1   +20.351, E3 +33195.219}
SPL {X  -160.000, Y  +607.824, Z    +0.000, E1   +20.354, E3 +33214.640}
SPL {X  -160.000, Y  +603.899, Z    +0.000, E1   +20.373, E3 +33237.090}
SPL {X  -160.000, Y  +599.617, Z    +0.000, E1   +20.384, E3 +33261.583}
SPL {X  -160.000, Y  +595.532, Z    +0.000, E1   +20.373, E3 +33284.944}
SPL {X  -160.000, Y  +591.705, Z    +0.000, E1   +20.373, E3 +33306.869}
SPL {X  -160.000, Y  +588.037, Z    +0.000, E1   +20.359, E3 +33327.956}
SPL {X  -160.000, Y  +584.320, Z    +0.000, E1   +20.364, E3 +33349.257}
SPL {X  -160.000, Y  +580.616, Z    +0.000, E1   +20.357, E3 +33370.484}
SPL {X  -160.000, Y  +577.083, Z    +0.000, E1   +20.358, E3 +33390.732}
SPL {X  -160.000, Y  +573.158, Z    +0.000, E1   +20.377, E3 +33413.185}
SPL {X  -160.000, Y  +568.802, Z    +0.000, E1   +20.385, E3 +33438.137}
SPL {X  -160.000, Y  +564.937, Z    +0.000, E1   +20.350, E3 +33460.357}
SPL {X  -160.000, Y  +561.213, Z    +0.000, E1   +20.372, E3 +33481.643}
SPL {X  -160.000, Y  +557.320, Z    +0.000, E1   +20.363, E3 +33503.970}
SPL {X  -160.000, Y  +553.712, Z    +0.000, E1   +20.355, E3 +33524.670}
SPL {X  -160.000, Y  +550.040, Z    +0.000, E1   +20.360, E3 +33545.708}
SPL {X  -160.000, Y  +546.180, Z    +0.000, E1   +20.370, E3 +33567.763}
SPL {X  -160.000, Y  +542.032, Z    +0.000, E1   +20.384, E3 +33591.502}
SPL {X  -160.000, Y  +537.870, Z    +0.000, E1   +20.372, E3 +33615.378}
SPL {X  -160.000, Y  +534.086, Z    +0.000, E1   +20.356, E3 +33637.132}
SPL {X  -160.000, Y  +530.164, Z    +0.000, E1   +20.382, E3 +33659.482}
SPL {X  -160.000, Y  +527.505, Z    +0.000, E1   +20.318, E3 +33674.855}
SPL {X  -160.000, Y  +511.620, Z    +0.000, E1   +28.365, E3 +33685.318}
SPL {X  -160.000, Y  +507.906, Z    +0.000, E1   +28.152, E3 +33701.713}
SPL {X  -160.000, Y  +506.085, Z    +0.000, E1   +26.146, E3 +33724.173}
SPL {X  -160.000, Y  +504.342, Z    +0.000, E1   +24.109, E3 +33747.688}
SPL {X  -160.000, Y  +503.002, Z    +0.000, E1   +22.325, E3 +33768.693}
SPL {X  -160.000, Y  +500.783, Z    +0.000, E1   +21.421, E3 +33788.283}
SPL {X  -160.000, Y  +497.229, Z    +0.000, E1   +21.403, E3 +33807.591}
SPL {X  -160.000, Y  +493.901, Z    +0.000, E1   +21.409, E3 +33825.610}
SPL {X  -160.000, Y  +490.791, Z    +0.000, E1   +21.400, E3 +33842.483}
SPL {X  -160.000, Y  +487.647, Z    +0.000, E1   +21.401, E3 +33859.529}
SPL {X  -160.000, Y  +484.273, Z    +0.000, E1   +21.408, E3 +33877.809}
SPL {X  -160.000, Y  +481.093, Z    +0.000, E1   +21.389, E3 +33895.118}
SPL {X  -160.000, Y  +478.021, Z    +0.000, E1   +21.401, E3 +33911.725}
SPL {X  -160.000, Y  +474.639, Z    +0.000, E1   +21.410, E3 +33930.016}
SPL {X  -160.000, Y  +471.343, Z    +0.000, E1   +21.399, E3 +33947.918}
SPL {X  -160.000, Y  +468.133, Z    +0.000, E1   +21.402, E3 +33965.309}
SPL {X  -160.000, Y  +464.638, Z    +0.000, E1   +21.421, E3 +33984.159}
SPL {X  -160.000, Y  +461.045, Z    +0.000, E1   +21.424, E3 +34003.572}
SPL {X  -160.000, Y  +457.606, Z    +0.000, E1   +21.413, E3 +34022.283}
SPL {X  -160.000, Y  +454.417, Z    +0.000, E1   +21.401, E3 +34039.591}
SPL {X  -160.000, Y  +451.425, Z    +0.000, E1   +21.404, E3 +34055.813}
SPL {X  -160.000, Y  +448.039, Z    +0.000, E1   +21.417, E3 +34074.105}
SPL {X  -160.000, Y  +444.787, Z    +0.000, E1   +21.414, E3 +34091.661}
SPL {X  -160.000, Y  +441.637, Z    +0.000, E1   +21.431, E3 +34108.639}
SPL {X  -160.000, Y  +438.199, Z    +0.000, E1   +21.432, E3 +34127.243}
SPL {X  -160.000, Y  +434.875, Z    +0.000, E1   +21.424, E3 +34145.283}
SPL {X  -160.000, Y  +431.689, Z    +0.000, E1   +21.423, E3 +34162.531}
SPL {X  -160.000, Y  +428.451, Z    +0.000, E1   +21.430, E3 +34180.010}
SPL {X  -160.000, Y  +425.120, Z    +0.000, E1   +21.430, E3 +34198.075}
SPL {X  -160.000, Y  +421.671, Z    +0.000, E1   +21.430, E3 +34216.759}
SPL {X  -160.000, Y  +418.225, Z    +0.000, E1   +21.425, E3 +34235.440}
SPL {X  -160.000, Y  +414.956, Z    +0.000, E1   +21.424, E3 +34253.121}
SPL {X  -160.000, Y  +411.834, Z    +0.000, E1   +21.420, E3 +34270.039}
SPL {X  -160.000, Y  +408.570, Z    +0.000, E1   +21.432, E3 +34287.648}
SPL {X  -160.000, Y  +405.237, Z    +0.000, E1   +21.432, E3 +34305.677}
SPL {X  -160.000, Y  +402.004, Z    +0.000, E1   +21.424, E3 +34323.252}
SPL {X  -160.000, Y  +398.626, Z    +0.000, E1   +21.425, E3 +34341.558}
SPL {X  -160.000, Y  +395.405, Z    +0.000, E1   +21.422, E3 +34358.976}
SPL {X  -160.000, Y  +392.641, Z    +0.000, E1   +21.407, E3 +34373.974}
SPL {X  -159.989, Y  +390.129, Z    +0.000, E1   +21.406, E3 +34387.615}
SPL {X  -159.932, Y  +387.337, Z    +0.000, E1   +21.403, E3 +34402.811}
SPL {X  -159.823, Y  +384.478, Z    +0.000, E1   +21.379, E3 +34418.474}
SPL {X  -159.660, Y  +381.581, Z    +0.000, E1   +21.363, E3 +34434.362}
SPL {X  -159.452, Y  +378.773, Z    +0.000, E1   +21.330, E3 +34449.809}
SPL {X  -159.222, Y  +376.244, Z    +0.000, E1   +21.297, E3 +34463.771}
SPL {X  -158.814, Y  +372.556, Z    +0.000, E1   +21.316, E3 +34484.038}
SPL {X  -158.301, Y  +368.743, Z    +0.000, E1   +21.199, E3 +34505.360}
SPL {X  -157.981, Y  +366.660, Z    +0.000, E1   +19.986, E3 +34528.327}
ENDSPLINE

SPLINE
SPL {X  -158.491, Y  +370.077, Z    +0.000, E1   +15.910, E3 +34553.341}
SPL {X  -159.771, Y  +383.450, Z    +0.000, E1    +6.314, E3 +34576.496}
SPL {X  -160.000, Y  +392.463, Z    +0.000, E1    +0.112, E3 +34583.003}
SPL {X  -160.000, Y  +399.874, Z    +0.000, E1    -5.508, E3 +34587.505}
SPL {X  -160.000, Y  +411.622, Z    +0.000, E1   -13.815, E3 +34599.625}
SPL {X  -160.000, Y  +419.836, Z    +0.000, E1   -18.198, E3 +34614.799}
SPL {X  -160.000, Y  +430.523, Z    +0.000, E1   -21.710, E3 +34644.999}
SPL {X  -160.000, Y  +433.426, Z    +0.000, E1   -21.735, E3 +34660.413}
SPL {X  -160.000, Y  +436.131, Z    +0.000, E1   -21.710, E3 +34674.888}
SPL {X  -160.000, Y  +439.046, Z    +0.000, E1   -21.732, E3 +34690.382}
SPL {X  -160.000, Y  +442.009, Z    +0.000, E1   -21.719, E3 +34706.204}
SPL {X  -160.000, Y  +444.891, Z    +0.000, E1   -21.724, E3 +34721.559}
SPL {X  -160.000, Y  +449.017, Z    +0.000, E1   -21.792, E3 +34743.351}
SPL {X  -160.000, Y  +452.864, Z    +0.000, E1   -21.730, E3 +34763.969}
SPL {X  -160.000, Y  +455.470, Z    +0.000, E1   -21.722, E3 +34777.858}
SPL {X  -160.000, Y  +458.295, Z    +0.000, E1   -21.738, E3 +34792.878}
SPL {X  -160.000, Y  +461.133, Z    +0.000, E1   -21.720, E3 +34808.061}
SPL {X  -160.000, Y  +464.458, Z    +0.000, E1   -21.770, E3 +34825.580}
SPL {X  -160.000, Y  +468.250, Z    +0.000, E1   -21.764, E3 +34845.733}
SPL {X  -160.000, Y  +472.226, Z    +0.000, E1   -21.782, E3 +34866.891}
SPL {X  -160.000, Y  +476.333, Z    +0.000, E1   -21.767, E3 +34888.806}
SPL {X  -160.000, Y  +480.244, Z    +0.000, E1   -21.765, E3 +34909.671}
SPL {X  -160.000, Y  +484.301, Z    +0.000, E1   -21.775, E3 +34931.199}
SPL {X  -160.000, Y  +488.201, Z    +0.000, E1   -21.768, E3 +34951.959}
SPL {X  -160.000, Y  +492.394, Z    +0.000, E1   -21.802, E3 +34974.133}
SPL {X  -160.000, Y  +496.781, Z    +0.000, E1   -21.798, E3 +34997.445}
SPL {X  -160.000, Y  +501.083, Z    +0.000, E1   -21.796, E3 +35020.374}
SPL {X  -160.000, Y  +504.917, Z    +0.000, E1   -21.764, E3 +35040.879}
SPL {X  -160.000, Y  +508.886, Z    +0.000, E1   -21.791, E3 +35061.965}
SPL {X  -160.000, Y  +513.057, Z    +0.000, E1   -21.767, E3 +35084.273}
SPL {X  -160.000, Y  +517.221, Z    +0.000, E1   -21.778, E3 +35106.425}
SPL {X  -160.000, Y  +521.677, Z    +0.000, E1   -21.781, E3 +35130.186}
SPL {X  -160.000, Y  +525.729, Z    +0.000, E1   -21.753, E3 +35151.826}
SPL {X  -160.000, Y  +529.456, Z    +0.000, E1   -21.766, E3 +35171.605}
SPL {X  -160.000, Y  +533.608, Z    +0.000, E1   -21.776, E3 +35193.736}
SPL {X  -160.000, Y  +538.227, Z    +0.000, E1   -21.794, E3 +35218.268}
SPL {X  -160.000, Y  +542.483, Z    +0.000, E1   -21.764, E3 +35240.993}
SPL {X  -160.000, Y  +546.194, Z    +0.000, E1   -21.754, E3 +35260.810}
SPL {X  -160.000, Y  +550.131, Z    +0.000, E1   -21.771, E3 +35281.745}
SPL {X  -160.000, Y  +554.462, Z    +0.000, E1   -21.777, E3 +35304.800}
SPL {X  -160.000, Y  +558.542, Z    +0.000, E1   -21.758, E3 +35326.572}
SPL {X  -160.000, Y  +562.615, Z    +0.000, E1   -21.776, E3 +35348.228}
SPL {X  -160.000, Y  +566.764, Z    +0.000, E1   -21.764, E3 +35370.353}
SPL {X  -160.000, Y  +570.657, Z    +0.000, E1   -21.758, E3 +35391.100}
SPL {X  -160.000, Y  +574.688, Z    +0.000, E1   -21.771, E3 +35412.543}
SPL {X  -160.000, Y  +578.864, Z    +0.000, E1   -21.770, E3 +35434.794}
SPL {X  -160.000, Y  +582.807, Z    +0.000, E1   -21.754, E3 +35455.848}
SPL {X  -160.000, Y  +586.993, Z    +0.000, E1   -21.779, E3 +35478.084}
SPL {X  -160.000, Y  +591.368, Z    +0.000, E1   -21.775, E3 +35501.371}
SPL {X  -160.000, Y  +595.703, Z    +0.000, E1   -21.775, E3 +35524.480}
SPL {X  -160.000, Y  +599.558, Z    +0.000, E1   -21.748, E3 +35545.057}
SPL {X  -160.000, Y  +603.126, Z    +0.000, E1   -21.757, E3 +35564.037}
SPL {X  -160.000, Y  +607.107, Z    +0.000, E1   -21.766, E3 +35585.262}
SPL {X  -160.000, Y  +611.246, Z    +0.000, E1   -21.760, E3 +35607.335}
SPL {X  -160.000, Y  +615.151, Z    +0.000, E1   -21.752, E3 +35628.149}
SPL {X  -160.000, Y  +618.728, Z    +0.000, E1   -21.747, E3 +35647.211}
SPL {X  -160.000, Y  +622.318, Z    +0.000, E1   -21.753, E3 +35666.326}
SPL {X  -160.000, Y  +625.877, Z    +0.000, E1   -21.745, E3 +35685.304}
SPL {X  -160.000, Y  +629.892, Z    +0.000, E1   -21.777, E3 +35706.628}
SPL {X  -160.000, Y  +634.024, Z    +0.000, E1   -21.756, E3 +35728.678}
SPL {X  -160.000, Y  +637.661, Z    +0.000, E1   -21.748, E3 +35748.069}
SPL {X  -160.000, Y  +641.244, Z    +0.000, E1   -21.752, E3 +35767.140}
SPL {X  -160.000, Y  +645.120, Z    +0.000, E1   -21.762, E3 +35787.772}
SPL {X  -160.000, Y  +649.214, Z    +0.000, E1   -21.766, E3 +35809.560}
SPL {X  -160.000, Y  +653.188, Z    +0.000, E1   -21.771, E3 +35830.623}
SPL {X  -160.000, Y  +656.905, Z    +0.000, E1   -21.769, E3 +35850.398}
SPL {X  -160.000, Y  +660.685, Z    +0.000, E1   -21.769, E3 +35870.566}
SPL {X  -160.000, Y  +664.985, Z    +0.000, E1   -21.790, E3 +35893.419}
SPL {X  -159.993, Y  +669.170, Z    +0.000, E1   -21.763, E3 +35915.777}
SPL {X  -159.916, Y  +672.869, Z    +0.000, E1   -21.755, E3 +35935.522}
SPL {X  -159.752, Y  +676.610, Z    +0.000, E1   -21.740, E3 +35955.597}
SPL {X  -159.478, Y  +680.618, Z    +0.000, E1   -21.719, E3 +35977.196}
SPL {X  -159.108, Y  +684.576, Z    +0.000, E1   -21.664, E3 +35998.665}
SPL {X  -158.638, Y  +688.530, Z    +0.000, E1   -21.617, E3 +36020.187}
SPL {X  -158.097, Y  +692.303, Z    +0.000, E1   -21.529, E3 +36040.905}
ENDSPLINE

SPLINE
SPL {X  -158.264, Y  +691.203, Z    +0.000, E1   -17.264, E3 +36077.650}
SPL {X  -159.000, Y  +685.560, Z    +0.000, E1   -12.398, E3 +36098.825}
SPL {X  -159.924, Y  +672.625, Z    +0.000, E1    -3.689, E3 +36113.843}
SPL {X  -160.000, Y  +663.203, Z    +0.000, E1    +3.155, E3 +36120.497}
SPL {X  -160.000, Y  +652.103, Z    +0.000, E1   +11.247, E3 +36132.167}
SPL {X  -160.000, Y  +641.822, Z    +0.000, E1   +17.059, E3 +36151.541}
SPL {X  -160.000, Y  +631.293, Z    +0.000, E1   +20.354, E3 +36185.420}
SPL {X  -160.000, Y  +627.542, Z    +0.000, E1   +20.380, E3 +36206.827}
SPL {X  -160.000, Y  +623.532, Z    +0.000, E1   +20.378, E3 +36229.793}
SPL {X  -160.000, Y  +619.329, Z    +0.000, E1   +20.391, E3 +36253.831}
SPL {X  -160.000, Y  +614.967, Z    +0.000, E1   +20.392, E3 +36278.810}
SPL {X  -160.000, Y  +611.206, Z    +0.000, E1   +20.351, E3 +36300.482}
SPL {X  -160.000, Y  +607.824, Z    +0.000, E1   +20.354, E3 +36319.903}
SPL {X  -160.000, Y  +603.899, Z    +0.000, E1   +20.373, E3 +36342.353}
SPL {X  -160.000, Y  +599.617, Z    +0.000, E1   +20.384, E3 +36366.847}
SPL {X  -160.000, Y  +595.532, Z    +0.000, E1   +20.373, E3 +36390.207}
SPL {X  -160.000, Y  +591.705, Z    +0.000, E1   +20.373, E3 +36412.132}
SPL {X  -160.000, Y  +588.037, Z    +0.000, E1   +20.359, E3 +36433.219}
SPL {X  -160.000, Y  +584.320, Z    +0.000, E1   +20.364, E3 +36454.521}
SPL {X  -160.000, Y  +580.616, Z    +0.000, E1   +20.357, E3 +36475.747}
SPL {X  -160.000, Y  +577.083, Z    +0.000, E1   +20.358, E3 +36495.996}
SPL {X  -160.000, Y  +573.158, Z    +0.000, E1   +20.377, E3 +36518.448}
SPL {X  -160.000, Y  +568.802, Z    +0.000, E1   +20.385, E3 +36543.400}
SPL {X  -160.000, Y  +564.937, Z    +0.000, E1   +20.350, E3 +36565.621}
SPL {X  -160.000, Y  +561.213, Z    +0.000, E1   +20.372, E3 +36586.907}
SPL {X  -160.000, Y  +557.320, Z    +0.000, E1   +20.363, E3 +36609.234}
SPL {X  -160.000, Y  +553.712, Z    +0.000, E1   +20.355, E3 +36629.933}
SPL {X  -160.000, Y  +550.040, Z    +0.000, E1   +20.360, E3 +36650.971}
SPL {X  -160.000, Y  +546.180, Z    +0.000, E1   +20.370, E3 +36673.027}
SPL {X  -160.000, Y  +542.032, Z    +0.000, E1   +20.384, E3 +36696.766}
SPL {X  -160.000, Y  +537.870, Z    +0.000, E1   +20.372, E3 +36720.642}
SPL {X  -160.000, Y  +534.086, Z    +0.000, E1   +20.356, E3 +36742.395}
SPL {X  -160.000, Y  +530.164, Z    +0.000, E1   +20.382, E3 +36764.745}
SPL {X  -160.000, Y  +527.505, Z    +0.000, E1   +20.318, E3 +36780.119}
SPL {X  -160.000, Y  +511.620, Z    +0.000, E1   +28.365, E3 +36790.582}
SPL {X  -160.000, Y  +507.906, Z    +0.000, E1   +28.152, E3 +36806.977}
SPL {X  -160.000, Y  +506.085, Z    +0.000, E1   +26.146, E3 +36829.436}
SPL {X  -160.000, Y  +504.342, Z    +0.000, E1   +24.109, E3 +36852.951}
SPL {X  -160.000, Y  +503.002, Z    +0.000, E1   +22.325, E3 +36873.957}
SPL {X  -160.000, Y  +500.783, Z    +0.000, E1   +21.421, E3 +36893.546}
SPL {X  -160.000, Y  +497.229, Z    +0.000, E1   +21.403, E3 +36912.854}
SPL {X  -160.000, Y  +493.901, Z    +0.000, E1   +21.409, E3 +36930.873}
SPL {X  -160.000, Y  +490.791, Z    +0.000, E1   +21.400, E3 +36947.746}
SPL {X  -160.000, Y  +487.647, Z    +0.000, E1   +21.401, E3 +36964.793}
SPL {X  -160.000, Y  +484.273, Z    +0.000, E1   +21.408, E3 +36983.072}
SPL {X  -160.000, Y  +481.093, Z    +0.000, E1   +21.389, E3 +37000.381}
SPL {X  -160.000, Y  +478.021, Z    +0.000, E1   +21.401, E3 +37016.988}
SPL {X  -160.000, Y  +474.639, Z    +0.000, E1   +21.410, E3 +37035.279}
SPL {X  -160.000, Y  +471.343, Z    +0.000, E1   +21.399, E3 +37053.181}
SPL {X  -160.000, Y  +468.133, Z    +0.000, E1   +21.402, E3 +37070.573}
SPL {X  -160.000, Y  +464.638, Z    +0.000, E1   +21.421, E3 +37089.422}
SPL {X  -160.000, Y  +461.045, Z    +0.000, E1   +21.424, E3 +37108.836}
SPL {X  -160.000, Y  +457.606, Z    +0.000, E1   +21.413, E3 +37127.546}
SPL {X  -160.000, Y  +454.417, Z    +0.000, E1   +21.401, E3 +37144.855}
SPL {X  -160.000, Y  +451.425, Z    +0.000, E1   +21.404, E3 +37161.076}
SPL {X  -160.000, Y  +448.039, Z    +0.000, E1   +21.417, E3 +37179.369}
SPL {X  -160.000, Y  +444.787, Z    +0.000, E1   +21.414, E3 +37196.924}
SPL {X  -160.000, Y  +441.637, Z    +0.000, E1   +21.431, E3 +37213.902}
SPL {X  -160.000, Y  +438.199, Z    +0.000, E1   +21.432, E3 +37232.506}
SPL {X  -160.000, Y  +434.875, Z    +0.000, E1   +21.424, E3 +37250.546}
SPL {X  -160.000, Y  +431.689, Z    +0.000, E1   +21.423, E3 +37267.794}
SPL {X  -160.000, Y  +428.451, Z    +0.000, E1   +21.430, E3 +37285.274}
SPL {X  -160.000, Y  +425.120, Z    +0.000, E1   +21.430, E3 +37303.338}
SPL {X  -160.000, Y  +421.671, Z    +0.000, E1   +21.430, E3 +37322.022}
SPL {X  -160.000, Y  +418.225, Z    +0.000, E1   +21.425, E3 +37340.704}
SPL {X  -160.000, Y  +414.956, Z    +0.000, E1   +21.424, E3 +37358.385}
SPL {X  -160.000, Y  +411.834, Z    +0.000, E1   +21.420, E3 +37375.303}
SPL {X  -160.000, Y  +408.570, Z    +0.000, E1   +21.432, E3 +37392.912}
SPL {X  -160.000, Y  +405.237, Z    +0.000, E1   +21.432, E3 +37410.940}
SPL {X  -160.000, Y  +402.004, Z    +0.000, E1   +21.424, E3 +37428.516}
SPL {X  -160.000, Y  +398.626, Z    +0.000, E1   +21.425, E3 +37446.822}
SPL {X  -160.000, Y  +395.405, Z    +0.000, E1   +21.422, E3 +37464.239}
SPL {X  -160.000, Y  +392.641, Z    +0.000, E1   +21.407, E3 +37479.237}
SPL {X  -159.989, Y  +390.129, Z    +0.000, E1   +21.406, E3 +37492.878}
SPL {X  -159.932, Y  +387.337, Z    +0.000, E1   +21.403, E3 +37508.074}
SPL {X  -159.823, Y  +384.478, Z    +0.000, E1   +21.379, E3 +37523.737}
SPL {X  -159.660, Y  +381.581, Z    +0.000, E1   +21.363, E3 +37539.625}
SPL {X  -159.452, Y  +378.773, Z    +0.000, E1   +21.330, E3 +37555.072}
SPL {X  -159.222, Y  +376.244, Z    +0.000, E1   +21.297, E3 +37569.034}
SPL {X  -158.814, Y  +372.556, Z    +0.000, E1   +21.316, E3 +37589.302}
SPL {X  -158.301, Y  +368.743, Z    +0.000, E1   +21.199, E3 +37610.624}
SPL {X  -157.981, Y  +366.660, Z    +0.000, E1   +19.986, E3 +37633.591}
ENDSPLINE

SPLINE
SPL {X  -158.491, Y  +370.077, Z    +0.000, E1   +15.910, E3 +37658.604}
SPL {X  -159.771, Y  +383.450, Z    +0.000, E1    +6.314, E3 +37681.759}
SPL {X  -160.000, Y  +392.463, Z    +0.000, E1    +0.112, E3 +37688.266}
SPL {X  -160.000, Y  +399.874, Z    +0.000, E1    -5.508, E3 +37692.769}
SPL {X  -160.000, Y  +411.622, Z    +0.000, E1   -13.815, E3 +37704.888}
SPL {X  -160.000, Y  +419.836, Z    +0.000, E1   -18.198, E3 +37720.062}
SPL {X  -160.000, Y  +430.523, Z    +0.000, E1   -21.710, E3 +37750.262}
SPL {X  -160.000, Y  +433.426, Z    +0.000, E1   -21.735, E3 +37765.677}
SPL {X  -160.000, Y  +436.131, Z    +0.000, E1   -21.710, E3 +37780.152}
SPL {X  -160.000, Y  +439.046, Z    +0.000, E1   -21.732, E3 +37795.645}
SPL {X  -160.000, Y  +442.009, Z    +0.000, E1   -21.719, E3 +37811.467}
SPL {X  -160.000, Y  +444.891, Z    +0.000, E1   -21.724, E3 +37826.823}
SPL {X  -160.000, Y  +449.017, Z    +0.000, E1   -21.792, E3 +37848.614}
SPL {X  -160.000, Y  +452.864, Z    +0.000, E1   -21.730, E3 +37869.232}
SPL {X  -160.000, Y  +455.470, Z    +0.000, E1   -21.722, E3 +37883.121}
SPL {X  -160.000, Y  +458.295, Z    +0.000, E1   -21.738, E3 +37898.142}
SPL {X  -160.000, Y  +461.133, Z    +0.000, E1   -21.720, E3 +37913.325}
SPL {X  -160.000, Y  +464.458, Z    +0.000, E1   -21.770, E3 +37930.843}
SPL {X  -160.000, Y  +468.250, Z    +0.000, E1   -21.764, E3 +37950.997}
SPL {X  -160.000, Y  +472.226, Z    +0.000, E1   -21.782, E3 +37972.155}
SPL {X  -160.000, Y  +476.333, Z    +0.000, E1   -21.767, E3 +37994.070}
SPL {X  -160.000, Y  +480.244, Z    +0.000, E1   -21.765, E3 +38014.934}
SPL {X  -160.000, Y  +484.301, Z    +0.000, E1   -21.775, E3 +38036.462}
SPL {X  -160.000, Y  +488.201, Z    +0.000, E1   -21.768, E3 +38057.222}
SPL {X  -160.000, Y  +492.394, Z    +0.000, E1   -21.802, E3 +38079.397}
SPL {X  -160.000, Y  +496.781, Z    +0.000, E1   -21.798, E3 +38102.708}
SPL {X  -160.000, Y  +501.083, Z    +0.000, E1   -21.796, E3 +38125.638}
SPL {X  -160.000, Y  +504.917, Z    +0.000, E1   -21.764, E3 +38146.142}
SPL {X  -160.000, Y  +508.886, Z    +0.000, E1   -21.791, E3 +38167.229}
SPL {X  -160.000, Y  +513.057, Z    +0.000, E1   -21.767, E3 +38189.536}
SPL {X  -160.000, Y  +517.221, Z    +0.000, E1   -21.778, E3 +38211.689}
SPL {X  -160.000, Y  +521.677, Z    +0.000, E1   -21.781, E3 +38235.450}
SPL {X  -160.000, Y  +525.729, Z    +0.000, E1   -21.753, E3 +38257.089}
SPL {X  -160.000, Y  +529.456, Z    +0.000, E1   -21.766, E3 +38276.869}
SPL {X  -160.000, Y  +533.608, Z    +0.000, E1   -21.776, E3 +38298.999}
SPL {X  -160.000, Y  +538.227, Z    +0.000, E1   -21.794, E3 +38323.531}
SPL {X  -160.000, Y  +542.483, Z    +0.000, E1   -21.764, E3 +38346.257}
SPL {X  -160.000, Y  +546.194, Z    +0.000, E1   -21.754, E3 +38366.073}
SPL {X  -160.000, Y  +550.131, Z    +0.000, E1   -21.771, E3 +38387.009}
SPL {X  -160.000, Y  +554.462, Z    +0.000, E1   -21.777, E3 +38410.063}
SPL {X  -160.000, Y  +558.542, Z    +0.000, E1   -21.758, E3 +38431.836}
SPL {X  -160.000, Y  +562.615, Z    +0.000, E1   -21.776, E3 +38453.491}
SPL {X  -160.000, Y  +566.764, Z    +0.000, E1   -21.764, E3 +38475.616}
SPL {X  -160.000, Y  +570.657, Z    +0.000, E1   -21.758, E3 +38496.364}
SPL {X  -160.000, Y  +574.688, Z    +0.000, E1   -21.771, E3 +38517.806}
SPL {X  -160.000, Y  +578.864, Z    +0.000, E1   -21.770, E3 +38540.057}
SPL {X  -160.000, Y  +582.807, Z    +0.000, E1   -21.754, E3 +38561.112}
SPL {X  -160.000, Y  +586.993, Z    +0.000, E1   -21.779, E3 +38583.347}
SPL {X  -160.000, Y  +591.368, Z    +0.000, E1   -21.775, E3 +38606.634}
SPL {X  -160.000, Y  +595.703, Z    +0.000, E1   -21.775, E3 +38629.744}
SPL {X  -160.000, Y  +599.558, Z    +0.000, E1   -21.748, E3 +38650.321}
SPL {X  -160.000, Y  +603.126, Z    +0.000, E1   -21.757, E3 +38669.301}
SPL {X  -160.000, Y  +607.107, Z    +0.000, E1   -21.766, E3 +38690.526}
SPL {X  -160.000, Y  +611.246, Z    +0.000, E1   -21.760, E3 +38712.599}
SPL {X  -160.000, Y  +615.151, Z    +0.000, E1   -21.752, E3 +38733.412}
SPL {X  -160.000, Y  +618.728, Z    +0.000, E1   -21.747, E3 +38752.475}
SPL {X  -160.000, Y  +622.318, Z    +0.000, E1   -21.753, E3 +38771.589}
SPL {X  -160.000, Y  +625.877, Z    +0.000, E1   -21.745, E3 +38790.568}
SPL {X  -160.000, Y  +629.892, Z    +0.000, E1   -21.777, E3 +38811.891}
SPL {X  -160.000, Y  +634.024, Z    +0.000, E1   -21.756, E3 +38833.942}
SPL {X  -160.000, Y  +637.661, Z    +0.000, E1   -21.748, E3 +38853.332}
SPL {X  -160.000, Y  +641.244, Z    +0.000, E1   -21.752, E3 +38872.403}
SPL {X  -160.000, Y  +645.120, Z    +0.000, E1   -21.762, E3 +38893.035}
SPL {X  -160.000, Y  +649.214, Z    +0.000, E1   -21.766, E3 +38914.824}
SPL {X  -160.000, Y  +653.188, Z    +0.000, E1   -21.771, E3 +38935.886}
SPL {X  -160.000, Y  +656.905, Z    +0.000, E1   -21.769, E3 +38955.661}
SPL {X  -160.000, Y  +660.685, Z    +0.000, E1   -21.769, E3 +38975.829}
SPL {X  -160.000, Y  +664.985, Z    +0.000, E1   -21.790, E3 +38998.682}
SPL {X  -159.993, Y  +669.170, Z    +0.000, E1   -21.763, E3 +39021.041}
SPL {X  -159.916, Y  +672.869, Z    +0.000, E1   -21.755, E3 +39040.786}
SPL {X  -159.752, Y  +676.610, Z    +0.000, E1   -21.740, E3 +39060.860}
SPL {X  -159.478, Y  +680.618, Z    +0.000, E1   -21.719, E3 +39082.460}
SPL {X  -159.108, Y  +684.576, Z    +0.000, E1   -21.664, E3 +39103.929}
SPL {X  -158.638, Y  +688.530, Z    +0.000, E1   -21.617, E3 +39125.451}
SPL {X  -158.097, Y  +692.303, Z    +0.000, E1   -21.529, E3 +39146.168}
ENDSPLINE

SPLINE
SPL {X  -158.264, Y  +691.203, Z    +0.000, E1   -17.264, E3 +39182.914}
SPL {X  -159.000, Y  +685.560, Z    +0.000, E1   -12.398, E3 +39204.089}
SPL {X  -159.924, Y  +672.625, Z    +0.000, E1    -3.689, E3 +39219.106}
SPL {X  -160.000, Y  +663.203, Z    +0.000, E1    +3.155, E3 +39225.761}
SPL {X  -160.000, Y  +652.103, Z    +0.000, E1   +11.247, E3 +39237.431}
SPL {X  -160.000, Y  +641.822, Z    +0.000, E1   +17.059, E3 +39256.804}
SPL {X  -160.000, Y  +631.293, Z    +0.000, E1   +20.354, E3 +39290.684}
SPL {X  -160.000, Y  +627.542, Z    +0.000, E1   +20.380, E3 +39312.091}
SPL {X  -160.000, Y  +623.532, Z    +0.000, E1   +20.378, E3 +39335.057}
SPL {X  -160.000, Y  +619.329, Z    +0.000, E1   +20.391, E3 +39359.094}
SPL {X  -160.000, Y  +614.967, Z    +0.000, E1   +20.392, E3 +39384.074}
SPL {X  -160.000, Y  +611.206, Z    +0.000, E1   +20.351, E3 +39405.746}
SPL {X  -160.000, Y  +607.824, Z    +0.000, E1   +20.354, E3 +39425.167}
SPL {X  -160.000, Y  +603.899, Z    +0.000, E1   +20.373, E3 +39447.617}
SPL {X  -160.000, Y  +599.617, Z    +0.000, E1   +20.384, E3 +39472.110}
SPL {X  -160.000, Y  +595.532, Z    +0.000, E1   +20.373, E3 +39495.471}
SPL {X  -160.000, Y  +591.705, Z    +0.000, E1   +20.373, E3 +39517.396}
SPL {X  -160.000, Y  +588.037, Z    +0.000, E1   +20.359, E3 +39538.483}
SPL {X  -160.000, Y  +584.320, Z    +0.000, E1   +20.364, E3 +39559.784}
SPL {X  -160.000, Y  +580.616, Z    +0.000, E1   +20.357, E3 +39581.011}
SPL {X  -160.000, Y  +577.083, Z    +0.000, E1   +20.358, E3 +39601.259}
SPL {X  -160.000, Y  +573.158, Z    +0.000, E1   +20.377, E3 +39623.712}
SPL {X  -160.000, Y  +568.802, Z    +0.000, E1   +20.385, E3 +39648.664}
SPL {X  -160.000, Y  +564.937, Z    +0.000, E1   +20.350, E3 +39670.884}
SPL {X  -160.000, Y  +561.213, Z    +0.000, E1   +20.372, E3 +39692.171}
SPL {X  -160.000, Y  +557.320, Z    +0.000, E1   +20.363, E3 +39714.497}
SPL {X  -160.000, Y  +553.712, Z    +0.000, E1   +20.355, E3 +39735.197}
SPL {X  -160.000, Y  +550.040, Z    +0.000, E1   +20.360, E3 +39756.235}
SPL {X  -160.000, Y  +546.180, Z    +0.000, E1   +20.370, E3 +39778.290}
SPL {X  -160.000, Y  +542.032, Z    +0.000, E1   +20.384, E3 +39802.029}
SPL {X  -160.000, Y  +537.870, Z    +0.000, E1   +20.372, E3 +39825.905}
SPL {X  -160.000, Y  +534.086, Z    +0.000, E1   +20.356, E3 +39847.659}
SPL {X  -160.000, Y  +530.164, Z    +0.000, E1   +20.382, E3 +39870.009}
SPL {X  -160.000, Y  +527.505, Z    +0.000, E1   +20.318, E3 +39885.382}
SPL {X  -160.000, Y  +511.620, Z    +0.000, E1   +28.365, E3 +39895.845}
SPL {X  -160.000, Y  +507.906, Z    +0.000, E1   +28.152, E3 +39912.240}
SPL {X  -160.000, Y  +506.085, Z    +0.000, E1   +26.146, E3 +39934.700}
SPL {X  -160.000, Y  +504.342, Z    +0.000, E1   +24.109, E3 +39958.215}
SPL {X  -160.000, Y  +503.002, Z    +0.000, E1   +22.325, E3 +39979.220}
SPL {X  -160.000, Y  +500.783, Z    +0.000, E1   +21.421, E3 +39998.810}
SPL {X  -160.000, Y  +497.229, Z    +0.000, E1   +21.403, E3 +40018.118}
SPL {X  -160.000, Y  +493.901, Z    +0.000, E1   +21.409, E3 +40036.137}
SPL {X  -160.000, Y  +490.791, Z    +0.000, E1   +21.400, E3 +40053.010}
SPL {X  -160.000, Y  +487.647, Z    +0.000, E1   +21.401, E3 +40070.056}
SPL {X  -160.000, Y  +484.273, Z    +0.000, E1   +21.408, E3 +40088.336}
SPL {X  -160.000, Y  +481.093, Z    +0.000, E1   +21.389, E3 +40105.645}
SPL {X  -160.000, Y  +478.021, Z    +0.000, E1   +21.401, E3 +40122.252}
SPL {X  -160.000, Y  +474.639, Z    +0.000, E1   +21.410, E3 +40140.543}
SPL {X  -160.000, Y  +471.343, Z    +0.000, E1   +21.399, E3 +40158.445}
SPL {X  -160.000, Y  +468.133, Z    +0.000, E1   +21.402, E3 +40175.836}
SPL {X  -160.000, Y  +464.638, Z    +0.000, E1   +21.421, E3 +40194.686}
SPL {X  -160.000, Y  +461.045, Z    +0.000, E1   +21.424, E3 +40214.099}
SPL {X  -160.000, Y  +457.606, Z    +0.000, E1   +21.413, E3 +40232.810}
SPL {X  -160.000, Y  +454.417, Z    +0.000, E1   +21.401, E3 +40250.118}
SPL {X  -160.000, Y  +451.425, Z    +0.000, E1   +21.404, E3 +40266.340}
SPL {X  -160.000, Y  +448.039, Z    +0.000, E1   +21.417, E3 +40284.633}
SPL {X  -160.000, Y  +444.787, Z    +0.000, E1   +21.414, E3 +40302.188}
SPL {X  -160.000, Y  +441.637, Z    +0.000, E1   +21.431, E3 +40319.166}
SPL {X  -160.000, Y  +438.199, Z    +0.000, E1   +21.432, E3 +40337.770}
SPL {X  -160.000, Y  +434.875, Z    +0.000, E1   +21.424, E3 +40355.810}
SPL {X  -160.000, Y  +431.689, Z    +0.000, E1   +21.423, E3 +40373.058}
SPL {X  -160.000, Y  +428.451, Z    +0.000, E1   +21.430, E3 +40390.537}
SPL {X  -160.000, Y  +425.120, Z    +0.000, E1   +21.430, E3 +40408.602}
SPL {X  -160.000, Y  +421.671, Z    +0.000, E1   +21.430, E3 +40427.286}
SPL {X  -160.000, Y  +418.225, Z    +0.000, E1   +21.425, E3 +40445.967}
SPL {X  -160.000, Y  +414.956, Z    +0.000, E1   +21.424, E3 +40463.648}
SPL {X  -160.000, Y  +411.834, Z    +0.000, E1   +21.420, E3 +40480.566}
SPL {X  -160.000, Y  +408.570, Z    +0.000, E1   +21.432, E3 +40498.175}
SPL {X  -160.000, Y  +405.237, Z    +0.000, E1   +21.432, E3 +40516.204}
SPL {X  -160.000, Y  +402.004, Z    +0.000, E1   +21.424, E3 +40533.779}
SPL {X  -160.000, Y  +398.626, Z    +0.000, E1   +21.425, E3 +40552.085}
SPL {X  -160.000, Y  +395.405, Z    +0.000, E1   +21.422, E3 +40569.503}
SPL {X  -160.000, Y  +392.641, Z    +0.000, E1   +21.407, E3 +40584.501}
SPL {X  -159.989, Y  +390.129, Z    +0.000, E1   +21.406, E3 +40598.142}
SPL {X  -159.932, Y  +387.337, Z    +0.000, E1   +21.403, E3 +40613.338}
SPL {X  -159.823, Y  +384.478, Z    +0.000, E1   +21.379, E3 +40629.001}
SPL {X  -159.660, Y  +381.581, Z    +0.000, E1   +21.363, E3 +40644.889}
SPL {X  -159.452, Y  +378.773, Z    +0.000, E1   +21.330, E3 +40660.336}
SPL {X  -159.222, Y  +376.244, Z    +0.000, E1   +21.297, E3 +40674.298}
SPL {X  -158.814, Y  +372.556, Z    +0.000, E1   +21.316, E3 +40694.565}
SPL {X  -158.301, Y  +368.743, Z    +0.000, E1   +21.199, E3 +40715.887}
SPL {X  -157.981, Y  +366.660, Z    +0.000, E1   +19.986, E3 +40738.854}
ENDSPLINE

SPLINE
SPL {X  -158.491, Y  +370.077, Z    +0.000, E1   +15.910, E3 +40763.868}
SPL {X  -159.771, Y  +383.450, Z    +0.000, E1    +6.314, E3 +40787.023}
SPL {X  -160.000, Y  +392.463, Z    +0.000, E1    +0.112, E3 +40793.530}
SPL {X  -160.000, Y  +399.874, Z    +0.000, E1    -5.508, E3 +40798.032}
SPL {X  -160.000, Y  +411.622, Z    +0.000, E1   -13.815, E3 +40810.152}
SPL {X  -160.000, Y  +419.836, Z    +0.000, E1   -18.198, E3 +40825.326}
SPL {X  -160.000, Y  +430.523, Z    +0.000, E1   -21.710, E3 +40855.526}
SPL {X  -160.000, Y  +433.426, Z    +0.000, E1   -21.735, E3 +40870.940}
SPL {X  -160.000, Y  +436.131, Z    +0.000, E1   -21.710, E3 +40885.415}
SPL {X  -160.000, Y  +439.046, Z    +0.000, E1   -21.732, E3 +40900.909}
SPL {X  -160.000, Y  +442.009, Z    +0.000, E1   -21.719, E3 +40916.731}
SPL {X  -160.000, Y  +444.891, Z    +0.000, E1   -21.724, E3 +40932.086}
SPL {X  -160.000, Y  +449.017, Z    +0.000, E1   -21.792, E3 +40953.878}
SPL {X  -160.000, Y  +452.864, Z    +0.000, E1   -21.730, E3 +40974.496}
SPL {X  -160.000, Y  +455.470, Z    +0.000, E1   -21.722, E3 +40988.385}
SPL {X  -160.000, Y  +458.295, Z    +0.000, E1   -21.738, E3 +41003.405}
SPL {X  -160.000, Y  +461.133, Z    +0.000, E1   -21.720, E3 +41018.588}
SPL {X  -160.000, Y  +464.458, Z    +0.000, E1   -21.770, E3 +41036.107}
SPL {X  -160.000, Y  +468.250, Z    +0.000, E1   -21.764, E3 +41056.260}
SPL {X  -160.000, Y  +472.226, Z    +0.000, E1   -21.782, E3 +41077.419}
SPL {X  -160.000, Y  +476.333, Z    +0.000, E1   -21.767, E3 +41099.333}
SPL {X  -160.000, Y  +480.244, Z    +0.000, E1   -21.765, E3 +41120.198}
SPL {X  -160.000, Y  +484.301, Z    +0.000, E1   -21.775, E3 +41141.726}
SPL {X  -160.000, Y  +488.201, Z    +0.000, E1   -21.768, E3 +41162.486}
SPL {X  -160.000, Y  +492.394, Z    +0.000, E1   -21.802, E3 +41184.660}
SPL {X  -160.000, Y  +496.781, Z    +0.000, E1   -21.798, E3 +41207.972}
SPL {X  -160.000, Y  +501.083, Z    +0.000, E1   -21.796, E3 +41230.902}
SPL {X  -160.000, Y  +504.917, Z    +0.000, E1   -21.764, E3 +41251.406}
SPL {X  -160.000, Y  +508.886, Z    +0.000, E1   -21.791, E3 +41272.492}
SPL {X  -160.000, Y  +513.057, Z    +0.000, E1   -21.767, E3 +41294.800}
SPL {X  -160.000, Y  +517.221, Z    +0.000, E1   -21.778, E3 +41316.952}
SPL {X  -160.000, Y  +521.677, Z    +0.000, E1   -21.781, E3 +41340.713}
SPL {X  -160.000, Y  +525.729, Z    +0.000, E1   -21.753, E3 +41362.353}
SPL {X  -160.000, Y  +529.456, Z    +0.000, E1   -21.766, E3 +41382.132}
SPL {X  -160.000, Y  +533.608, Z    +0.000, E1   -21.776, E3 +41404.263}
SPL {X  -160.000, Y  +538.227, Z    +0.000, E1   -21.794, E3 +41428.795}
SPL {X  -160.000, Y  +542.483, Z    +0.000, E1   -21.764, E3 +41451.520}
SPL {X  -160.000, Y  +546.194, Z    +0.000, E1   -21.754, E3 +41471.337}
SPL {X  -160.000, Y  +550.131, Z    +0.000, E1   -21.771, E3 +41492.272}
SPL {X  -160.000, Y  +554.462, Z    +0.000, E1   -21.777, E3 +41515.327}
SPL {X  -160.000, Y  +558.542, Z    +0.000, E1   -21.758, E3 +41537.099}
SPL {X  -160.000, Y  +562.615, Z    +0.000, E1   -21.776, E3 +41558.755}
SPL {X  -160.000, Y  +566.764, Z    +0.000, E1   -21.764, E3 +41580.880}
SPL {X  -160.000, Y  +570.657, Z    +0.000, E1   -21.758, E3 +41601.627}
SPL {X  -160.000, Y  +574.688, Z    +0.000, E1   -21.771, E3 +41623.070}
SPL {X  -160.000, Y  +578.864, Z    +0.000, E1   -21.770, E3 +41645.321}
SPL {X  -160.000, Y  +582.807, Z    +0.000, E1   -21.754, E3 +41666.375}
SPL {X  -160.000, Y  +586.993, Z    +0.000, E1   -21.779, E3 +41688.611}
SPL {X  -160.000, Y  +591.368, Z    +0.000, E1   -21.775, E3 +41711.898}
SPL {X  -160.000, Y  +595.703, Z    +0.000, E1   -21.775, E3 +41735.007}
SPL {X  -160.000, Y  +599.558, Z    +0.000, E1   -21.748, E3 +41755.585}
SPL {X  -160.000, Y  +603.126, Z    +0.000, E1   -21.757, E3 +41774.564}
SPL {X  -160.000, Y  +607.107, Z    +0.000, E1   -21.766, E3 +41795.789}
SPL {X  -160.000, Y  +611.246, Z    +0.000, E1   -21.760, E3 +41817.862}
SPL {X  -160.000, Y  +615.151, Z    +0.000, E1   -21.752, E3 +41838.676}
SPL {X  -160.000, Y  +618.728, Z    +0.000, E1   -21.747, E3 +41857.738}
SPL {X  -160.000, Y  +622.318, Z    +0.000, E1   -21.753, E3 +41876.853}
SPL {X  -160.000, Y  +625.877, Z    +0.000, E1   -21.745, E3 +41895.831}
SPL {X  -160.000, Y  +629.892, Z    +0.000, E1   -21.777, E3 +41917.155}
SPL {X  -160.000, Y  +634.024, Z    +0.000, E1   -21.756, E3 +41939.205}
SPL {X  -160.000, Y  +637.661, Z    +0.000, E1   -21.748, E3 +41958.596}
SPL {X  -160.000, Y  +641.244, Z    +0.000, E1   -21.752, E3 +41977.667}
SPL {X  -160.000, Y  +645.120, Z    +0.000, E1   -21.762, E3 +41998.299}
SPL {X  -160.000, Y  +649.214, Z    +0.000, E1   -21.766, E3 +42020.087}
SPL {X  -160.000, Y  +653.188, Z    +0.000, E1   -21.771, E3 +42041.150}
SPL {X  -160.000, Y  +656.905, Z    +0.000, E1   -21.769, E3 +42060.925}
SPL {X  -160.000, Y  +660.685, Z    +0.000, E1   -21.769, E3 +42081.093}
SPL {X  -160.000, Y  +664.985, Z    +0.000, E1   -21.790, E3 +42103.946}
SPL {X  -159.993, Y  +669.170, Z    +0.000, E1   -21.763, E3 +42126.304}
SPL {X  -159.916, Y  +672.869, Z    +0.000, E1   -21.755, E3 +42146.049}
SPL {X  -159.752, Y  +676.610, Z    +0.000, E1   -21.740, E3 +42166.124}
SPL {X  -159.478, Y  +680.618, Z    +0.000, E1   -21.719, E3 +42187.723}
SPL {X  -159.108, Y  +684.576, Z    +0.000, E1   -21.664, E3 +42209.192}
SPL {X  -158.638, Y  +688.530, Z    +0.000, E1   -21.617, E3 +42230.714}
SPL {X  -158.097, Y  +692.303, Z    +0.000, E1   -21.529, E3 +42251.432}
ENDSPLINE

SPLINE
SPL {X  -158.264, Y  +691.203, Z    +0.000, E1   -17.264, E3 +42288.177}
SPL {X  -159.000, Y  +685.560, Z    +0.000, E1   -12.398, E3 +42309.352}
SPL {X  -159.924, Y  +672.625, Z    +0.000, E1    -3.689, E3 +42324.370}
SPL {X  -160.000, Y  +663.203, Z    +0.000, E1    +3.155, E3 +42331.024}
SPL {X  -160.000, Y  +652.103, Z    +0.000, E1   +11.247, E3 +42342.694}
SPL {X  -160.000, Y  +641.822, Z    +0.000, E1   +17.059, E3 +42362.068}
SPL {X  -160.000, Y  +631.293, Z    +0.000, E1   +20.354, E3 +42395.947}
SPL {X  -160.000, Y  +627.542, Z    +0.000, E1   +20.380, E3 +42417.355}
SPL {X  -160.000, Y  +623.532, Z    +0.000, E1   +20.378, E3 +42440.320}
SPL {X  -160.000, Y  +619.329, Z    +0.000, E1   +20.391, E3 +42464.358}
SPL {X  -160.000, Y  +614.967, Z    +0.000, E1   +20.392, E3 +42489.337}
SPL {X  -160.000, Y  +611.206, Z    +0.000, E1   +20.351, E3 +42511.009}
SPL {X  -160.000, Y  +607.824, Z    +0.000, E1   +20.354, E3 +42530.430}
SPL {X  -160.000, Y  +603.899, Z    +0.000, E1   +20.373, E3 +42552.880}
SPL {X  -160.000, Y  +599.617, Z    +0.000, E1   +20.384, E3 +42577.374}
SPL {X  -160.000, Y  +595.532, Z    +0.000, E1   +20.373, E3 +42600.734}
SPL {X  -160.000, Y  +591.705, Z    +0.000, E1   +20.373, E3 +42622.659}
SPL {X  -160.000, Y  +588.037, Z    +0.000, E1   +20.359, E3 +42643.746}
SPL {X  -160.000, Y  +584.320, Z    +0.000, E1   +20.364, E3 +42665.048}
SPL {X  -160.000, Y  +580.616, Z    +0.000, E1   +20.357, E3 +42686.274}
SPL {X  -160.000, Y  +577.083, Z    +0.000, E1   +20.358, E3 +42706.523}
SPL {X  -160.000, Y  +573.158, Z    +0.000, E1   +20.377, E3 +42728.975}
SPL {X  -160.000, Y  +568.802, Z    +0.000, E1   +20.385, E3 +42753.927}
SPL {X  -160.000, Y  +564.937, Z    +0.000, E1   +20.350, E3 +42776.148}
SPL {X  -160.000, Y  +561.213, Z    +0.000, E1   +20.372, E3 +42797.434}
SPL {X  -160.000, Y  +557.320, Z    +0.000, E1   +20.363, E3 +42819.761}
SPL {X  -160.000, Y  +553.712, Z    +0.000, E1   +20.355, E3 +42840.460}
SPL {X  -160.000, Y  +550.040, Z    +0.000, E1   +20.360, E3 +42861.498}
SPL {X  -160.000, Y  +546.180, Z    +0.000, E1   +20.370, E3 +42883.554}
SPL {X  -160.000, Y  +542.032, Z    +0.000, E1   +20.384, E3 +42907.293}
SPL {X  -160.000, Y  +537.870, Z    +0.000, E1   +20.372, E3 +42931.169}
SPL {X  -160.000, Y  +534.086, Z    +0.000, E1   +20.356, E3 +42952.922}
SPL {X  -160.000, Y  +530.164, Z    +0.000, E1   +20.382, E3 +42975.272}
SPL {X  -160.000, Y  +527.505, Z    +0.000, E1   +20.318, E3 +42990.646}
SPL {X  -160.000, Y  +511.620, Z    +0.000, E1   +28.365, E3 +43001.109}
SPL {X  -160.000, Y  +507.906, Z    +0.000, E1   +28.152, E3 +43017.504}
SPL {X  -160.000, Y  +506.085, Z    +0.000, E1   +26.146, E3 +43039.964}
SPL {X  -160.000, Y  +504.342, Z    +0.000, E1   +24.109, E3 +43063.479}
SPL {X  -160.000, Y  +503.002, Z    +0.000, E1   +22.325, E3 +43084.484}
SPL {X  -160.000, Y  +500.783, Z    +0.000, E1   +21.421, E3 +43104.073}
SPL {X  -160.000, Y  +497.229, Z    +0.000, E1   +21.403, E3 +43123.381}
SPL {X  -160.000, Y  +493.901, Z    +0.000, E1   +21.409, E3 +43141.400}
SPL {X  -160.000, Y  +490.791, Z    +0.000, E1   +21.400, E3 +43158.273}
SPL {X  -160.000, Y  +487.647, Z    +0.000, E1   +21.401, E3 +43175.320}
SPL {X  -160.000, Y  +484.273, Z    +0.000, E1   +21.408, E3 +43193.599}
SPL {X  -160.000, Y  +481.093, Z    +0.000, E1   +21.389, E3 +43210.909}
SPL {X  -160.000, Y  +478.021, Z    +0.000, E1   +21.401, E3 +43227.515}
SPL {X  -160.000, Y  +474.639, Z    +0.000, E1   +21.410, E3 +43245.806}
SPL {X  -160.000, Y  +471.343, Z    +0.000, E1   +21.399, E3 +43263.708}
SPL {X  -160.000, Y  +468.133, Z    +0.000, E1   +21.402, E3 +43281.100}
SPL {X  -160.000, Y  +464.638, Z    +0.000, E1   +21.421, E3 +43299.949}
SPL {X  -160.000, Y  +461.045, Z    +0.000, E1   +21.424, E3 +43319.363}
SPL {X  -160.000, Y  +457.606, Z    +0.000, E1   +21.413, E3 +43338.073}
SPL {X  -160.000, Y  +454.417, Z    +0.000, E1   +21.401, E3 +43355.382}
SPL {X  -160.000, Y  +451.425, Z    +0.000, E1   +21.404, E3 +43371.603}
SPL {X  -160.000, Y  +448.039, Z    +0.000, E1   +21.417, E3 +43389.896}
SPL {X  -160.000, Y  +444.787, Z    +0.000, E1   +21.414, E3 +43407.451}
SPL {X  -160.000, Y  +441.637, Z    +0.000, E1   +21.431, E3 +43424.429}
SPL {X  -160.000, Y  +438.199, Z    +0.000, E1   +21.432, E3 +43443.033}
SPL {X  -160.000, Y  +434.875, Z    +0.000, E1   +21.424, E3 +43461.073}
SPL {X  -160.000, Y  +431.689, Z    +0.000, E1   +21.423, E3 +43478.321}
SPL {X  -160.000, Y  +428.451, Z    +0.000, E1   +21.430, E3 +43495.801}
SPL {X  -160.000, Y  +425.120, Z    +0.000, E1   +21.430, E3 +43513.865}
SPL {X  -160.000, Y  +421.671, Z    +0.000, E1   +21.430, E3 +43532.549}
SPL {X  -160.000, Y  +418.225, Z    +0.000, E1   +21.425, E3 +43551.231}
SPL {X  -160.000, Y  +414.956, Z    +0.000, E1   +21.424, E3 +43568.912}
SPL {X  -160.000, Y  +411.834, Z    +0.000, E1   +21.420, E3 +43585.830}
SPL {X  -160.000, Y  +408.570, Z    +0.000, E1   +21.432, E3 +43603.439}
SPL {X  -160.000, Y  +405.237, Z    +0.000, E1   +21.432, E3 +43621.467}
SPL {X  -160.000, Y  +402.004, Z    +0.000, E1   +21.424, E3 +43639.043}
SPL {X  -160.000, Y  +398.626, Z    +0.000, E1   +21.425, E3 +43657.349}
SPL {X  -160.000, Y  +395.405, Z    +0.000, E1   +21.422, E3 +43674.766}
SPL {X  -160.000, Y  +392.641, Z    +0.000, E1   +21.407, E3 +43689.765}
SPL {X  -159.989, Y  +390.129, Z    +0.000, E1   +21.406, E3 +43703.405}
SPL {X  -159.932, Y  +387.337, Z    +0.000, E1   +21.403, E3 +43718.601}
SPL {X  -159.823, Y  +384.478, Z    +0.000, E1   +21.379, E3 +43734.264}
SPL {X  -159.660, Y  +381.581, Z    +0.000, E1   +21.363, E3 +43750.152}
SPL {X  -159.452, Y  +378.773, Z    +0.000, E1   +21.330, E3 +43765.599}
SPL {X  -159.222, Y  +376.244, Z    +0.000, E1   +21.297, E3 +43779.561}
SPL {X  -158.814, Y  +372.556, Z    +0.000, E1   +21.316, E3 +43799.829}
SPL {X  -158.301, Y  +368.743, Z    +0.000, E1   +21.199, E3 +43821.151}
SPL {X  -157.981, Y  +366.660, Z    +0.000, E1   +19.986, E3 +43844.118}
ENDSPLINE

SPLINE
SPL {X  -158.491, Y  +370.077, Z    +0.000, E1   +15.910, E3 +43869.131}
SPL {X  -159.771, Y  +383.450, Z    +0.000, E1    +6.314, E3 +43892.286}
SPL {X  -160.000, Y  +392.463, Z    +0.000, E1    +0.112, E3 +43898.793}
SPL {X  -160.000, Y  +399.874, Z    +0.000, E1    -5.508, E3 +43903.296}
SPL {X  -160.000, Y  +411.622, Z    +0.000, E1   -13.815, E3 +43915.415}
SPL {X  -160.000, Y  +419.836, Z    +0.000, E1   -18.198, E3 +43930.589}
SPL {X  -160.000, Y  +430.523, Z    +0.000, E1   -21.710, E3 +43960.789}
SPL {X  -160.000, Y  +433.426, Z    +0.000, E1   -21.735, E3 +43976.204}
SPL {X  -160.000, Y  +436.131, Z    +0.000, E1   -21.710, E3 +43990.679}
SPL {X  -160.000, Y  +439.046, Z    +0.000, E1   -21.732, E3 +44006.172}
SPL {X  -160.000, Y  +442.009, Z    +0.000, E1   -21.719, E3 +44021.994}
SPL {X  -160.000, Y  +444.891, Z    +0.000, E1   -21.724, E3 +44037.350}
SPL {X  -160.000, Y  +449.017, Z    +0.000, E1   -21.792, E3 +44059.141}
SPL {X  -160.000, Y  +452.864, Z    +0.000, E1   -21.730, E3 +44079.759}
SPL {X  -160.000, Y  +455.470, Z    +0.000, E1   -21.722, E3 +44093.648}
SPL {X  -160.000, Y  +458.295, Z    +0.000, E1   -21.738, E3 +44108.669}
SPL {X  -160.000, Y  +461.133, Z    +0.000, E1   -21.720, E3 +44123.852}
SPL {X  -160.000, Y  +464.458, Z    +0.000, E1   -21.770, E3 +44141.370}
SPL {X  -160.000, Y  +468.250, Z    +0.000, E1   -21.764, E3 +44161.524}
SPL {X  -160.000, Y  +472.226, Z    +0.000, E1   -21.782, E3 +44182.682}
SPL {X  -160.000, Y  +476.333, Z    +0.000, E1   -21.767, E3 +44204.597}
SPL {X  -160.000, Y  +480.244, Z    +0.000, E1   -21.765, E3 +44225.461}
SPL {X  -160.000, Y  +484.301, Z    +0.000, E1   -21.775, E3 +44246.990}
SPL {X  -160.000, Y  +488.201, Z    +0.000, E1   -21.768, E3 +44267.749}
SPL {X  -160.000, Y  +492.394, Z    +0.000, E1   -21.802, E3 +44289.924}
SPL {X  -160.000, Y  +496.781, Z    +0.000, E1   -21.798, E3 +44313.235}
SPL {X  -160.000, Y  +501.083, Z    +0.000, E1   -21.796, E3 +44336.165}
SPL {X  -160.000, Y  +504.917, Z    +0.000, E1   -21.764, E3 +44356.670}
SPL {X  -160.000, Y  +508.886, Z    +0.000, E1   -21.791, E3 +44377.756}
SPL {X  -160.000, Y  +513.057, Z    +0.000, E1   -21.767, E3 +44400.063}
SPL {X  -160.000, Y  +517.221, Z    +0.000, E1   -21.778, E3 +44422.216}
SPL {X  -160.000, Y  +521.677, Z    +0.000, E1   -21.781, E3 +44445.977}
SPL {X  -160.000, Y  +525.729, Z    +0.000, E1   -21.753, E3 +44467.616}
SPL {X  -160.000, Y  +529.456, Z    +0.000, E1   -21.766, E3 +44487.396}
SPL {X  -160.000, Y  +533.608, Z    +0.000, E1   -21.776, E3 +44509.526}
SPL {X  -160.000, Y  +538.227, Z    +0.000, E1   -21.794, E3 +44534.059}
SPL {X  -160.000, Y  +542.483, Z    +0.000, E1   -21.764, E3 +44556.784}
SPL {X  -160.000, Y  +546.194, Z    +0.000, E1   -21.754, E3 +44576.600}
SPL {X  -160.000, Y  +550.131, Z    +0.000, E1   -21.771, E3 +44597.536}
SPL {X  -160.000, Y  +554.462, Z    +0.000, E1   -21.777, E3 +44620.590}
SPL {X  -160.000, Y  +558.542, Z    +0.000, E1   -21.758, E3 +44642.363}
SPL {X  -160.000, Y  +562.615, Z    +0.000, E1   -21.776, E3 +44664.018}
SPL {X  -160.000, Y  +566.764, Z    +0.000, E1   -21.764, E3 +44686.143}
SPL {X  -160.000, Y  +570.657, Z    +0.000, E1   -21.758, E3 +44706.891}
SPL {X  -160.000, Y  +574.688, Z    +0.000, E1   -21.771, E3 +44728.333}
SPL {X  -160.000, Y  +578.864, Z    +0.000, E1   -21.770, E3 +44750.584}
SPL {X  -160.000, Y  +582.807, Z    +0.000, E1   -21.754, E3 +44771.639}
SPL {X  -160.000, Y  +586.993, Z    +0.000, E1   -21.779, E3 +44793.874}
SPL {X  -160.000, Y  +591.368, Z    +0.000, E1   -21.775, E3 +44817.161}
SPL {X  -160.000, Y  +595.703, Z    +0.000, E1   -21.775, E3 +44840.271}
SPL {X  -160.000, Y  +599.558, Z    +0.000, E1   -21.748, E3 +44860.848}
SPL {X  -160.000, Y  +603.126, Z    +0.000, E1   -21.757, E3 +44879.828}
SPL {X  -160.000, Y  +607.107, Z    +0.000, E1   -21.766, E3 +44901.053}
SPL {X  -160.000, Y  +611.246, Z    +0.000, E1   -21.760, E3 +44923.126}
SPL {X  -160.000, Y  +615.151, Z    +0.000, E1   -21.752, E3 +44943.939}
SPL {X  -160.000, Y  +618.728, Z    +0.000, E1   -21.747, E3 +44963.002}
SPL {X  -160.000, Y  +622.318, Z    +0.000, E1   -21.753, E3 +44982.116}
SPL {X  -160.000, Y  +625.877, Z    +0.000, E1   -21.745, E3 +45001.095}
SPL {X  -160.000, Y  +629.892, Z    +0.000, E1   -21.777, E3 +45022.418}
SPL {X  -160.000, Y  +634.024, Z    +0.000, E1   -21.756, E3 +45044.469}
SPL {X  -160.000, Y  +637.661, Z    +0.000, E1   -21.748, E3 +45063.859}
SPL {X  -160.000, Y  +641.244, Z    +0.000, E1   -21.752, E3 +45082.930}
SPL {X  -160.000, Y  +645.120, Z    +0.000, E1   -21.762, E3 +45103.562}
SPL {X  -160.000, Y  +649.214, Z    +0.000, E1   -21.766, E3 +45125.351}
SPL {X  -160.000, Y  +653.188, Z    +0.000, E1   -21.771, E3 +45146.413}
SPL {X  -160.000, Y  +656.905, Z    +0.000, E1   -21.769, E3 +45166.188}
SPL {X  -160.000, Y  +660.685, Z    +0.000, E1   -21.769, E3 +45186.356}
SPL {X  -160.000, Y  +664.985, Z    +0.000, E1   -21.790, E3 +45209.209}
SPL {X  -159.993, Y  +669.170, Z    +0.000, E1   -21.763, E3 +45231.568}
SPL {X  -159.916, Y  +672.869, Z    +0.000, E1   -21.755, E3 +45251.313}
SPL {X  -159.752, Y  +676.610, Z    +0.000, E1   -21.740, E3 +45271.387}
SPL {X  -159.478, Y  +680.618, Z    +0.000, E1   -21.719, E3 +45292.987}
SPL {X  -159.108, Y  +684.576, Z    +0.000, E1   -21.664, E3 +45314.456}
SPL {X  -158.638, Y  +688.530, Z    +0.000, E1   -21.617, E3 +45335.978}
SPL {X  -158.097, Y  +692.303, Z    +0.000, E1   -21.529, E3 +45356.695}
ENDSPLINE

SPLINE
SPL {X  -158.264, Y  +691.203, Z    +0.000, E1   -17.264, E3 +45393.441}
SPL {X  -159.000, Y  +685.560, Z    +0.000, E1   -12.398, E3 +45414.616}
SPL {X  -159.924, Y  +672.625, Z    +0.000, E1    -3.689, E3 +45429.633}
SPL {X  -160.000, Y  +663.203, Z    +0.000, E1    +3.155, E3 +45436.288}
SPL {X  -160.000, Y  +652.103, Z    +0.000, E1   +11.247, E3 +45447.958}
SPL {X  -160.000, Y  +641.822, Z    +0.000, E1   +17.059, E3 +45467.332}
SPL {X  -160.000, Y  +631.293, Z    +0.000, E1   +20.354, E3 +45501.211}
SPL {X  -160.000, Y  +627.542, Z    +0.000, E1   +20.380, E3 +45522.618}
SPL {X  -160.000, Y  +623.532, Z    +0.000, E1   +20.378, E3 +45545.584}
SPL {X  -160.000, Y  +619.329, Z    +0.000, E1   +20.391, E3 +45569.621}
SPL {X  -160.000, Y  +614.967, Z    +0.000, E1   +20.392, E3 +45594.601}
SPL {X  -160.000, Y  +611.206, Z    +0.000, E1   +20.351, E3 +45616.273}
SPL {X  -160.000, Y  +607.824, Z    +0.000, E1   +20.354, E3 +45635.694}
SPL {X  -160.000, Y  +603.899, Z    +0.000, E1   +20.373, E3 +45658.144}
SPL {X  -160.000, Y  +599.617, Z    +0.000, E1   +20.384, E3 +45682.637}
SPL {X  -160.000, Y  +595.532, Z    +0.000, E1   +20.373, E3 +45705.998}
SPL {X  -160.000, Y  +591.705, Z    +0.000, E1   +20.373, E3 +45727.923}
SPL {X  -160.000, Y  +588.037, Z    +0.000, E1   +20.359, E3 +45749.010}
SPL {X  -160.000, Y  +584.320, Z    +0.000, E1   +20.364, E3 +45770.311}
SPL {X  -160.000, Y  +580.616, Z    +0.000, E1   +20.357, E3 +45791.538}
SPL {X  -160.000, Y  +577.083, Z    +0.000, E1   +20.358, E3 +45811.787}
SPL {X  -160.000, Y  +573.158, Z    +0.000, E1   +20.377, E3 +45834.239}
SPL {X  -160.000, Y  +568.802, Z    +0.000, E1   +20.385, E3 +45859.191}
SPL {X  -160.000, Y  +564.937, Z    +0.000, E1   +20.350, E3 +45881.411}
SPL {X  -160.000, Y  +561.213, Z    +0.000, E1   +20.372, E3 +45902.698}
SPL {X  -160.000, Y  +557.320, Z    +0.000, E1   +20.363, E3 +45925.024}
SPL {X  -160.000, Y  +553.712, Z    +0.000, E1   +20.355, E3 +45945.724}
SPL {X  -160.000, Y  +550.040, Z    +0.000, E1   +20.360, E3 +45966.762}
SPL {X  -160.000, Y  +546.180, Z    +0.000, E1   +20.370, E3 +45988.817}
SPL {X  -160.000, Y  +542.032, Z    +0.000, E1   +20.384, E3 +46012.557}
SPL {X  -160.000, Y  +537.870, Z    +0.000, E1   +20.372, E3 +46036.432}
SPL {X  -160.000, Y  +534.086, Z    +0.000, E1   +20.356, E3 +46058.186}
SPL {X  -160.000, Y  +530.164, Z    +0.000, E1   +20.382, E3 +46080.536}
SPL {X  -160.000, Y  +527.505, Z    +0.000, E1   +20.318, E3 +46095.909}
SPL {X  -160.000, Y  +511.620, Z    +0.000, E1   +28.365, E3 +46106.372}
SPL {X  -160.000, Y  +507.906, Z    +0.000, E1   +28.152, E3 +46122.768}
SPL {X  -160.000, Y  +506.085, Z    +0.000, E1   +26.146, E3 +46145.227}
SPL {X  -160.000, Y  +504.342, Z    +0.000, E1   +24.109, E3 +46168.742}
SPL {X  -160.000, Y  +503.002, Z    +0.000, E1   +22.325, E3 +46189.748}
SPL {X  -160.000, Y  +500.783, Z    +0.000, E1   +21.421, E3 +46209.337}
SPL {X  -160.000, Y  +497.229, Z    +0.000, E1   +21.403, E3 +46228.645}
SPL {X  -160.000, Y  +493.901, Z    +0.000, E1   +21.409, E3 +46246.664}
SPL {X  -160.000, Y  +490.791, Z    +0.000, E1   +21.400, E3 +46263.537}
SPL {X  -160.000, Y  +487.647, Z    +0.000, E1   +21.401, E3 +46280.583}
SPL {X  -160.000, Y  +484.273, Z    +0.000, E1   +21.408, E3 +46298.863}
SPL {X  -160.000, Y  +481.093, Z    +0.000, E1   +21.389, E3 +46316.172}
SPL {X  -160.000, Y  +478.021, Z    +0.000, E1   +21.401, E3 +46332.779}
SPL {X  -160.000, Y  +474.639, Z    +0.000, E1   +21.410, E3 +46351.070}
SPL {X  -160.000, Y  +471.343, Z    +0.000, E1   +21.399, E3 +46368.972}
SPL {X  -160.000, Y  +468.133, Z    +0.000, E1   +21.402, E3 +46386.364}
SPL {X  -160.000, Y  +464.638, Z    +0.000, E1   +21.421, E3 +46405.213}
SPL {X  -160.000, Y  +461.045, Z    +0.000, E1   +21.424, E3 +46424.626}
SPL {X  -160.000, Y  +457.606, Z    +0.000, E1   +21.413, E3 +46443.337}
SPL {X  -160.000, Y  +454.417, Z    +0.000, E1   +21.401, E3 +46460.645}
SPL {X  -160.000, Y  +451.425, Z    +0.000, E1   +21.404, E3 +46476.867}
SPL {X  -160.000, Y  +448.039, Z    +0.000, E1   +21.417, E3 +46495.160}
SPL {X  -160.000, Y  +444.787, Z    +0.000, E1   +21.414, E3 +46512.715}
SPL {X  -160.000, Y  +441.637, Z    +0.000, E1   +21.431, E3 +46529.693}
SPL {X  -160.000, Y  +438.199, Z    +0.000, E1   +21.432, E3 +46548.297}
SPL {X  -160.000, Y  +434.875, Z    +0.000, E1   +21.424, E3 +46566.337}
SPL {X  -160.000, Y  +431.689, Z    +0.000, E1   +21.423, E3 +46583.585}
SPL {X  -160.000, Y  +428.451, Z    +0.000, E1   +21.430, E3 +46601.064}
SPL {X  -160.000, Y  +425.120, Z    +0.000, E1   +21.430, E3 +46619.129}
SPL {X  -160.000, Y  +421.671, Z    +0.000, E1   +21.430, E3 +46637.813}
SPL {X  -160.000, Y  +418.225, Z    +0.000, E1   +21.425, E3 +46656.494}
SPL {X  -160.000, Y  +414.956, Z    +0.000, E1   +21.424, E3 +46674.175}
SPL {X  -160.000, Y  +411.834, Z    +0.000, E1   +21.420, E3 +46691.093}
SPL {X  -160.000, Y  +408.570, Z    +0.000, E1   +21.432, E3 +46708.702}
SPL {X  -160.000, Y  +405.237, Z    +0.000, E1   +21.432, E3 +46726.731}
SPL {X  -160.000, Y  +402.004, Z    +0.000, E1   +21.424, E3 +46744.306}
SPL {X  -160.000, Y  +398.626, Z    +0.000, E1   +21.425, E3 +46762.612}
SPL {X  -160.000, Y  +395.405, Z    +0.000, E1   +21.422, E3 +46780.030}
SPL {X  -160.000, Y  +392.641, Z    +0.000, E1   +21.407, E3 +46795.028}
SPL {X  -159.989, Y  +390.129, Z    +0.000, E1   +21.406, E3 +46808.669}
SPL {X  -159.932, Y  +387.337, Z    +0.000, E1   +21.403, E3 +46823.865}
SPL {X  -159.823, Y  +384.478, Z    +0.000, E1   +21.379, E3 +46839.528}
SPL {X  -159.660, Y  +381.581, Z    +0.000, E1   +21.363, E3 +46855.416}
SPL {X  -159.452, Y  +378.773, Z    +0.000, E1   +21.330, E3 +46870.863}
SPL {X  -159.222, Y  +376.244, Z    +0.000, E1   +21.297, E3 +46884.825}
SPL {X  -158.814, Y  +372.556, Z    +0.000, E1   +21.316, E3 +46905.092}
SPL {X  -158.301, Y  +368.743, Z    +0.000, E1   +21.199, E3 +46926.414}
SPL {X  -157.981, Y  +366.660, Z    +0.000, E1   +19.986, E3 +46949.382}
ENDSPLINE

SPLINE
SPL {X  -158.491, Y  +370.077, Z    +0.000, E1   +15.910, E3 +46974.395}
SPL {X  -159.771, Y  +383.450, Z    +0.000, E1    +6.314, E3 +46997.550}
SPL {X  -160.000, Y  +392.463, Z    +0.000, E1    +0.112, E3 +47004.057}
SPL {X  -160.000, Y  +399.874, Z    +0.000, E1    -5.508, E3 +47008.559}
SPL {X  -160.000, Y  +411.622, Z    +0.000, E1   -13.815, E3 +47020.679}
SPL {X  -160.000, Y  +419.836, Z    +0.000, E1   -18.198, E3 +47035.853}
SPL {X  -160.000, Y  +430.523, Z    +0.000, E1   -21.710, E3 +47066.053}
SPL {X  -160.000, Y  +433.426, Z    +0.000, E1   -21.735, E3 +47081.467}
SPL {X  -160.000, Y  +436.131, Z    +0.000, E1   -21.710, E3 +47095.942}
SPL {X  -160.000, Y  +439.046, Z    +0.000, E1   -21.732, E3 +47111.436}
SPL {X  -160.000, Y  +442.009, Z    +0.000, E1   -21.719, E3 +47127.258}
SPL {X  -160.000, Y  +444.891, Z    +0.000, E1   -21.724, E3 +47142.613}
SPL {X  -160.000, Y  +449.017, Z    +0.000, E1   -21.792, E3 +47164.405}
SPL {X  -160.000, Y  +452.864, Z    +0.000, E1   -21.730, E3 +47185.023}
SPL {X  -160.000, Y  +455.470, Z    +0.000, E1   -21.722, E3 +47198.912}
SPL {X  -160.000, Y  +458.295, Z    +0.000, E1   -21.738, E3 +47213.932}
SPL {X  -160.000, Y  +461.133, Z    +0.000, E1   -21.720, E3 +47229.115}
SPL {X  -160.000, Y  +464.458, Z    +0.000, E1   -21.770, E3 +47246.634}
SPL {X  -160.000, Y  +468.250, Z    +0.000, E1   -21.764, E3 +47266.787}
SPL {X  -160.000, Y  +472.226, Z    +0.000, E1   -21.782, E3 +47287.946}
SPL {X  -160.000, Y  +476.333, Z    +0.000, E1   -21.767, E3 +47309.860}
SPL {X  -160.000, Y  +480.244, Z    +0.000, E1   -21.765, E3 +47330.725}
SPL {X  -160.000, Y  +484.301, Z    +0.000, E1   -21.775, E3 +47352.253}
SPL {X  -160.000, Y  +488.201, Z    +0.000, E1   -21.768, E3 +47373.013}
SPL {X  -160.000, Y  +492.394, Z    +0.000, E1   -21.802, E3 +47395.187}
SPL {X  -160.000, Y  +496.781, Z    +0.000, E1   -21.798, E3 +47418.499}
SPL {X  -160.000, Y  +501.083, Z    +0.000, E1   -21.796, E3 +47441.429}
SPL {X  -160.000, Y  +504.917, Z    +0.000, E1   -21.764, E3 +47461.933}
SPL {X  -160.000, Y  +508.886, Z    +0.000, E1   -21.791, E3 +47483.019}
SPL {X  -160.000, Y  +513.057, Z    +0.000, E1   -21.767, E3 +47505.327}
SPL {X  -160.000, Y  +517.221, Z    +0.000, E1   -21.778, E3 +47527.479}
SPL {X  -160.000, Y  +521.677, Z    +0.000, E1   -21.781, E3 +47551.240}
SPL {X  -160.000, Y  +525.729, Z    +0.000, E1   -21.753, E3 +47572.880}
SPL {X  -160.000, Y  +529.456, Z    +0.000, E1   -21.766, E3 +47592.659}
SPL {X  -160.000, Y  +533.608, Z    +0.000, E1   -21.776, E3 +47614.790}
SPL {X  -160.000, Y  +538.227, Z    +0.000, E1   -21.794, E3 +47639.322}
SPL {X  -160.000, Y  +542.483, Z    +0.000, E1   -21.764, E3 +47662.047}
SPL {X  -160.000, Y  +546.194, Z    +0.000, E1   -21.754, E3 +47681.864}
SPL {X  -160.000, Y  +550.131, Z    +0.000, E1   -21.771, E3 +47702.800}
SPL {X  -160.000, Y  +554.462, Z    +0.000, E1   -21.777, E3 +47725.854}
SPL {X  -160.000, Y  +558.542, Z    +0.000, E1   -21.758, E3 +47747.626}
SPL {X  -160.000, Y  +562.615, Z    +0.000, E1   -21.776, E3 +47769.282}
SPL {X  -160.000, Y  +566.764, Z    +0.000, E1   -21.764, E3 +47791.407}
SPL {X  -160.000, Y  +570.657, Z    +0.000, E1   -21.758, E3 +47812.154}
SPL {X  -160.000, Y  +574.688, Z    +0.000, E1   -21.771, E3 +47833.597}
SPL {X  -160.000, Y  +578.864, Z    +0.000, E1   -21.770, E3 +47855.848}
SPL {X  -160.000, Y  +582.807, Z    +0.000, E1   -21.754, E3 +47876.902}
SPL {X  -160.000, Y  +586.993, Z    +0.000, E1   -21.779, E3 +47899.138}
SPL {X  -160.000, Y  +591.368, Z    +0.000, E1   -21.775, E3 +47922.425}
SPL {X  -160.000, Y  +595.703, Z    +0.000, E1   -21.775, E3 +47945.534}
SPL {X  -160.000, Y  +599.558, Z    +0.000, E1   -21.748, E3 +47966.112}
SPL {X  -160.000, Y  +603.126, Z    +0.000, E1   -21.757, E3 +47985.091}
SPL {X  -160.000, Y  +607.107, Z    +0.000, E1   -21.766, E3 +48006.316}
SPL {X  -160.000, Y  +611.246, Z    +0.000, E1   -21.760, E3 +48028.390}
SPL {X  -160.000, Y  +615.151, Z    +0.000, E1   -21.752, E3 +48049.203}
SPL {X  -160.000, Y  +618.728, Z    +0.000, E1   -21.747, E3 +48068.265}
SPL {X  -160.000, Y  +622.318, Z    +0.000, E1   -21.753, E3 +48087.380}
SPL {X  -160.000, Y  +625.877, Z    +0.000, E1   -21.745, E3 +48106.358}
SPL {X  -160.000, Y  +629.892, Z    +0.000, E1   -21.777, E3 +48127.682}
SPL {X  -160.000, Y  +634.024, Z    +0.000, E1   -21.756, E3 +48149.732}
SPL {X  -160.000, Y  +637.661, Z    +0.000, E1   -21.748, E3 +48169.123}
SPL {X  -160.000, Y  +641.244, Z    +0.000, E1   -21.752, E3 +48188.194}
SPL {X  -160.000, Y  +645.120, Z    +0.000, E1   -21.762, E3 +48208.826}
SPL {X  -160.000, Y  +649.214, Z    +0.000, E1   -21.766, E3 +48230.614}
SPL {X  -160.000, Y  +653.188, Z    +0.000, E1   -21.771, E3 +48251.677}
SPL {X  -160.000, Y  +656.905, Z    +0.000, E1   -21.769, E3 +48271.452}
SPL {X  -160.000, Y  +660.685, Z    +0.000, E1   -21.769, E3 +48291.620}
SPL {X  -160.000, Y  +664.985, Z    +0.000, E1   -21.790, E3 +48314.473}
SPL {X  -159.993, Y  +669.170, Z    +0.000, E1   -21.763, E3 +48336.831}
SPL {X  -159.916, Y  +672.869, Z    +0.000, E1   -21.755, E3 +48356.576}
SPL {X  -159.752, Y  +676.610, Z    +0.000, E1   -21.740, E3 +48376.651}
SPL {X  -159.478, Y  +680.618, Z    +0.000, E1   -21.719, E3 +48398.250}
SPL {X  -159.108, Y  +684.576, Z    +0.000, E1   -21.664, E3 +48419.720}
SPL {X  -158.638, Y  +688.530, Z    +0.000, E1   -21.617, E3 +48441.241}
SPL {X  -158.097, Y  +692.303, Z    +0.000, E1   -21.529, E3 +48461.959}
ENDSPLINE

SPLINE
SPL {X  -158.264, Y  +691.203, Z    +0.000, E1   -17.264, E3 +48498.704}
SPL {X  -159.000, Y  +685.560, Z    +0.000, E1   -12.398, E3 +48519.880}
SPL {X  -159.924, Y  +672.625, Z    +0.000, E1    -3.689, E3 +48534.897}
SPL {X  -160.000, Y  +663.203, Z    +0.000, E1    +3.155, E3 +48541.551}
SPL {X  -160.000, Y  +652.103, Z    +0.000, E1   +11.247, E3 +48553.221}
SPL {X  -160.000, Y  +641.822, Z    +0.000, E1   +17.059, E3 +48572.595}
SPL {X  -160.000, Y  +631.293, Z    +0.000, E1   +20.354, E3 +48606.474}
SPL {X  -160.000, Y  +627.542, Z    +0.000, E1   +20.380, E3 +48627.882}
SPL {X  -160.000, Y  +623.532, Z    +0.000, E1   +20.378, E3 +48650.847}
SPL {X  -160.000, Y  +619.329, Z    +0.000, E1   +20.391, E3 +48674.885}
SPL {X  -160.000, Y  +614.967, Z    +0.000, E1   +20.392, E3 +48699.865}
SPL {X  -160.000, Y  +611.206, Z    +0.000, E1   +20.351, E3 +48721.536}
SPL {X  -160.000, Y  +607.824, Z    +0.000, E1   +20.354, E3 +48740.957}
SPL {X  -160.000, Y  +603.899, Z    +0.000, E1   +20.373, E3 +48763.407}
SPL {X  -160.000, Y  +599.617, Z    +0.000, E1   +20.384, E3 +48787.901}
SPL {X  -160.000, Y  +595.532, Z    +0.000, E1   +20.373, E3 +48811.261}
SPL {X  -160.000, Y  +591.705, Z    +0.000, E1   +20.373, E3 +48833.186}
SPL {X  -160.000, Y  +588.037, Z    +0.000, E1   +20.359, E3 +48854.273}
SPL {X  -160.000, Y  +584.320, Z    +0.000, E1   +20.364, E3 +48875.575}
SPL {X  -160.000, Y  +580.616, Z    +0.000, E1   +20.357, E3 +48896.802}
SPL {X  -160.000, Y  +577.083, Z    +0.000, E1   +20.358, E3 +48917.050}
SPL {X  -160.000, Y  +573.158, Z    +0.000, E1   +20.377, E3 +48939.502}
SPL {X  -160.000, Y  +568.802, Z    +0.000, E1   +20.385, E3 +48964.454}
SPL {X  -160.000, Y  +564.937, Z    +0.000, E1   +20.350, E3 +48986.675}
SPL {X  -160.000, Y  +561.213, Z    +0.000, E1   +20.372, E3 +49007.961}
SPL {X  -160.000, Y  +557.320, Z    +0.000, E1   +20.363, E3 +49030.288}
SPL {X  -160.000, Y  +553.712, Z    +0.000, E1   +20.355, E3 +49050.987}
SPL {X  -160.000, Y  +550.040, Z    +0.000, E1   +20.360, E3 +49072.025}
SPL {X  -160.000, Y  +546.180, Z    +0.000, E1   +20.370, E3 +49094.081}
SPL {X  -160.000, Y  +542.032, Z    +0.000, E1   +20.384, E3 +49117.820}
SPL {X  -160.000, Y  +537.870, Z    +0.000, E1   +20.372, E3 +49141.696}
SPL {X  -160.000, Y  +534.086, Z    +0.000, E1   +20.356, E3 +49163.449}
SPL {X  -160.000, Y  +530.164, Z    +0.000, E1   +20.382, E3 +49185.799}
SPL {X  -160.000, Y  +527.505, Z    +0.000, E1   +20.318, E3 +49201.173}
SPL {X  -160.000, Y  +511.620, Z    +0.000, E1   +28.365, E3 +49211.636}
SPL {X  -160.000, Y  +507.906, Z    +0.000, E1   +28.152, E3 +49228.031}
SPL {X  -160.000, Y  +506.085, Z    +0.000, E1   +26.146, E3 +49250.491}
SPL {X  -160.000, Y  +504.342, Z    +0.000, E1   +24.109, E3 +49274.006}
SPL {X  -160.000, Y  +503.002, Z    +0.000, E1   +22.325, E3 +49295.011}
SPL {X  -160.000, Y  +500.783, Z    +0.000, E1   +21.421, E3 +49314.600}
SPL {X  -160.000, Y  +497.229, Z    +0.000, E1   +21.403, E3 +49333.908}
SPL {X  -160.000, Y  +493.901, Z    +0.000, E1   +21.409, E3 +49351.927}
SPL {X  -160.000, Y  +490.791, Z    +0.000, E1   +21.400, E3 +49368.800}
SPL {X  -160.000, Y  +487.647, Z    +0.000, E1   +21.401, E3 +49385.847}
SPL {X  -160.000, Y  +484.273, Z    +0.000, E1   +21.408, E3 +49404.126}
SPL {X  -160.000, Y  +481.093, Z    +0.000, E1   +21.389, E3 +49421.436}
SPL {X  -160.000, Y  +478.021, Z    +0.000, E1   +21.401, E3 +49438.042}
SPL {X  -160.000, Y  +474.639, Z    +0.000, E1   +21.410, E3 +49456.333}
SPL {X  -160.000, Y  +471.343, Z    +0.000, E1   +21.399, E3 +49474.236}
SPL {X  -160.000, Y  +468.133, Z    +0.000, E1   +21.402, E3 +49491.627}
SPL {X  -160.000, Y  +464.638, Z    +0.000, E1   +21.421, E3 +49510.476}
SPL {X  -160.000, Y  +461.045, Z    +0.000, E1   +21.424, E3 +49529.890}
SPL {X  -160.000, Y  +457.606, Z    +0.000, E1   +21.413, E3 +49548.600}
SPL {X  -160.000, Y  +454.417, Z    +0.000, E1   +21.401, E3 +49565.909}
SPL {X  -160.000, Y  +451.425, Z    +0.000, E1   +21.404, E3 +49582.130}
SPL {X  -160.000, Y  +448.039, Z    +0.000, E1   +21.417, E3 +49600.423}
SPL {X  -160.000, Y  +444.787, Z    +0.000, E1   +21.414, E3 +49617.978}
SPL {X  -160.000, Y  +441.637, Z    +0.000, E1   +21.431, E3 +49634.956}
SPL {X  -160.000, Y  +438.199, Z    +0.000, E1   +21.432, E3 +49653.560}
SPL {X  -160.000, Y  +434.875, Z    +0.000, E1   +21.424, E3 +49671.600}
SPL {X  -160.000, Y  +431.689, Z    +0.000, E1   +21.423, E3 +49688.848}
SPL {X  -160.000, Y  +428.451, Z    +0.000, E1   +21.430, E3 +49706.328}
SPL {X  -160.000, Y  +425.120, Z    +0.000, E1   +21.430, E3 +49724.392}
SPL {X  -160.000, Y  +421.671, Z    +0.000, E1   +21.430, E3 +49743.076}
SPL {X  -160.000, Y  +418.225, Z    +0.000, E1   +21.425, E3 +49761.758}
SPL {X  -160.000, Y  +414.956, Z    +0.000, E1   +21.424, E3 +49779.439}
SPL {X  -160.000, Y  +411.834, Z    +0.000, E1   +21.420, E3 +49796.357}
SPL {X  -160.000, Y  +408.570, Z    +0.000, E1   +21.432, E3 +49813.966}
SPL {X  -160.000, Y  +405.237, Z    +0.000, E1   +21.432, E3 +49831.994}
SPL {X  -160.000, Y  +402.004, Z    +0.000, E1   +21.424, E3 +49849.570}
SPL {X  -160.000, Y  +398.626, Z    +0.000, E1   +21.425, E3 +49867.876}
SPL {X  -160.000, Y  +395.405, Z    +0.000, E1   +21.422, E3 +49885.293}
SPL {X  -160.000, Y  +392.641, Z    +0.000, E1   +21.407, E3 +49900.292}
SPL {X  -159.989, Y  +390.129, Z    +0.000, E1   +21.406, E3 +49913.932}
SPL {X  -159.932, Y  +387.337, Z    +0.000, E1   +21.403, E3 +49929.128}
SPL {X  -159.823, Y  +384.478, Z    +0.000, E1   +21.379, E3 +49944.791}
SPL {X  -159.660, Y  +381.581, Z    +0.000, E1   +21.363, E3 +49960.679}
SPL {X  -159.452, Y  +378.773, Z    +0.000, E1   +21.330, E3 +49976.126}
SPL {X  -159.222, Y  +376.244, Z    +0.000, E1   +21.297, E3 +49990.088}
SPL {X  -158.814, Y  +372.556, Z    +0.000, E1   +21.316, E3 +50010.356}
SPL {X  -158.301, Y  +368.743, Z    +0.000, E1   +21.199, E3 +50031.678}
SPL {X  -157.981, Y  +366.660, Z    +0.000, E1   +19.986, E3 +50054.645}
ENDSPLINE

SPLINE
SPL {X  -158.491, Y  +370.077, Z    +0.000, E1   +15.910, E3 +50079.658}
SPL {X  -159.771, Y  +383.450, Z    +0.000, E1    +6.314, E3 +50102.813}
SPL {X  -160.000, Y  +392.463, Z    +0.000, E1    +0.112, E3 +50109.320}
SPL {X  -160.000, Y  +399.874, Z    +0.000, E1    -5.508, E3 +50113.823}
SPL {X  -160.000, Y  +411.622, Z    +0.000, E1   -13.815, E3 +50125.942}
SPL {X  -160.000, Y  +419.836, Z    +0.000, E1   -18.198, E3 +50141.116}
SPL {X  -160.000, Y  +430.523, Z    +0.000, E1   -21.710, E3 +50171.316}
SPL {X  -160.000, Y  +433.426, Z    +0.000, E1   -21.735, E3 +50186.731}
SPL {X  -160.000, Y  +436.131, Z    +0.000, E1   -21.710, E3 +50201.206}
SPL {X  -160.000, Y  +439.046, Z    +0.000, E1   -21.732, E3 +50216.699}
SPL {X  -160.000, Y  +442.009, Z    +0.000, E1   -21.719, E3 +50232.521}
SPL {X  -160.000, Y  +444.891, Z    +0.000, E1   -21.724, E3 +50247.877}
SPL {X  -160.000, Y  +449.017, Z    +0.000, E1   -21.792, E3 +50269.669}
SPL {X  -160.000, Y  +452.864, Z    +0.000, E1   -21.730, E3 +50290.286}
SPL {X  -160.000, Y  +455.470, Z    +0.000, E1   -21.722, E3 +50304.175}
SPL {X  -160.000, Y  +458.295, Z    +0.000, E1   -21.738, E3 +50319.196}
SPL {X  -160.000, Y  +461.133, Z    +0.000, E1   -21.720, E3 +50334.379}
SPL {X  -160.000, Y  +464.458, Z    +0.000, E1   -21.770, E3 +50351.897}
SPL {X  -160.000, Y  +468.250, Z    +0.000, E1   -21.764, E3 +50372.051}
SPL {X  -160.000, Y  +472.226, Z    +0.000, E1   -21.782, E3 +50393.209}
SPL {X  -160.000, Y  +476.333, Z    +0.000, E1   -21.767, E3 +50415.124}
SPL {X  -160.000, Y  +480.244, Z    +0.000, E1   -21.765, E3 +50435.988}
SPL {X  -160.000, Y  +484.301, Z    +0.000, E1   -21.775, E3 +50457.517}
SPL {X  -160.000, Y  +488.201, Z    +0.000, E1   -21.768, E3 +50478.276}
SPL {X  -160.000, Y  +492.394, Z    +0.000, E1   -21.802, E3 +50500.451}
SPL {X  -160.000, Y  +496.781, Z    +0.000, E1   -21.798, E3 +50523.762}
SPL {X  -160.000, Y  +501.083, Z    +0.000, E1   -21.796, E3 +50546.692}
SPL {X  -160.000, Y  +504.917, Z    +0.000, E1   -21.764, E3 +50567.197}
SPL {X  -160.000, Y  +508.886, Z    +0.000, E1   -21.791, E3 +50588.283}
SPL {X  -160.000, Y  +513.057, Z    +0.000, E1   -21.767, E3 +50610.590}
SPL {X  -160.000, Y  +517.221, Z    +0.000, E1   -21.778, E3 +50632.743}
SPL {X  -160.000, Y  +521.677, Z    +0.000, E1   -21.781, E3 +50656.504}
SPL {X  -160.000, Y  +525.729, Z    +0.000, E1   -21.753, E3 +50678.143}
SPL {X  -160.000, Y  +529.456, Z    +0.000, E1   -21.766, E3 +50697.923}
SPL {X  -160.000, Y  +533.608, Z    +0.000, E1   -21.776, E3 +50720.053}
SPL {X  -160.000, Y  +538.227, Z    +0.000, E1   -21.794, E3 +50744.586}
SPL {X  -160.000, Y  +542.483, Z    +0.000, E1   -21.764, E3 +50767.311}
SPL {X  -160.000, Y  +546.194, Z    +0.000, E1   -21.754, E3 +50787.127}
SPL {X  -160.000, Y  +550.131, Z    +0.000, E1   -21.771, E3 +50808.063}
SPL {X  -160.000, Y  +554.462, Z    +0.000, E1   -21.777, E3 +50831.117}
SPL {X  -160.000, Y  +558.542, Z    +0.000, E1   -21.758, E3 +50852.890}
SPL {X  -160.000, Y  +562.615, Z    +0.000, E1   -21.776, E3 +50874.545}
SPL {X  -160.000, Y  +566.764, Z    +0.000, E1   -21.764, E3 +50896.670}
SPL {X  -160.000, Y  +570.657, Z    +0.000, E1   -21.758, E3 +50917.418}
SPL {X  -160.000, Y  +574.688, Z    +0.000, E1   -21.771, E3 +50938.861}
SPL {X  -160.000, Y  +578.864, Z    +0.000, E1   -21.770, E3 +50961.111}
SPL {X  -160.000, Y  +582.807, Z    +0.000, E1   -21.754, E3 +50982.166}
SPL {X  -160.000, Y  +586.993, Z    +0.000, E1   -21.779, E3 +51004.401}
SPL {X  -160.000, Y  +591.368, Z    +0.000, E1   -21.775, E3 +51027.688}
SPL {X  -160.000, Y  +595.703, Z    +0.000, E1   -21.775, E3 +51050.798}
SPL {X  -160.000, Y  +599.558, Z    +0.000, E1   -21.748, E3 +51071.375}
SPL {X  -160.000, Y  +603.126, Z    +0.000, E1   -21.757, E3 +51090.355}
SPL {X  -160.000, Y  +607.107, Z    +0.000, E1   -21.766, E3 +51111.580}
SPL {X  -160.000, Y  +611.246, Z    +0.000, E1   -21.760, E3 +51133.653}
SPL {X  -160.000, Y  +615.151, Z    +0.000, E1   -21.752, E3 +51154.466}
SPL {X  -160.000, Y  +618.728, Z    +0.000, E1   -21.747, E3 +51173.529}
SPL {X  -160.000, Y  +622.318, Z    +0.000, E1   -21.753, E3 +51192.643}
SPL {X  -160.000, Y  +625.877, Z    +0.000, E1   -21.745, E3 +51211.622}
SPL {X  -160.000, Y  +629.892, Z    +0.000, E1   -21.777, E3 +51232.945}
SPL {X  -160.000, Y  +634.024, Z    +0.000, E1   -21.756, E3 +51254.996}
SPL {X  -160.000, Y  +637.661, Z    +0.000, E1   -21.748, E3 +51274.386}
SPL {X  -160.000, Y  +641.244, Z    +0.000, E1   -21.752, E3 +51293.457}
SPL {X  -160.000, Y  +645.120, Z    +0.000, E1   -21.762, E3 +51314.089}
SPL {X  -160.000, Y  +649.214, Z    +0.000, E1   -21.766, E3 +51335.878}
SPL {X  -160.000, Y  +653.188, Z    +0.000, E1   -21.771, E3 +51356.940}
SPL {X  -160.000, Y  +656.905, Z    +0.000, E1   -21.769, E3 +51376.716}
SPL {X  -160.000, Y  +660.685, Z    +0.000, E1   -21.769, E3 +51396.883}
SPL {X  -160.000, Y  +664.985, Z    +0.000, E1   -21.790, E3 +51419.736}
SPL {X  -159.993, Y  +669.170, Z    +0.000, E1   -21.763, E3 +51442.095}
SPL {X  -159.916, Y  +672.869, Z    +0.000, E1   -21.755, E3 +51461.840}
SPL {X  -159.752, Y  +676.610, Z    +0.000, E1   -21.740, E3 +51481.914}
SPL {X  -159.478, Y  +680.618, Z    +0.000, E1   -21.719, E3 +51503.514}
SPL {X  -159.108, Y  +684.576, Z    +0.000, E1   -21.664, E3 +51524.983}
SPL {X  -158.638, Y  +688.530, Z    +0.000, E1   -21.617, E3 +51546.505}
SPL {X  -158.097, Y  +692.303, Z    +0.000, E1   -21.529, E3 +51567.222}
ENDSPLINE

